// TwinCAT 3 PLC project Fraktal_Core
// Title: Fraktal_Core
// Company: fraktal-automation
// Author: fraktal-automation
// ProjectVersion: 0.1.0.3
// Description: Fraktal Core framework library: contracts, base classes (CM/EM/Unit), PermIntlk, profiler, connector base, recipe provider (Core 2.2).
// ProgramVersion: 3.1.4024.0
// libraries:
//   Tc2_Standard, * (Beckhoff Automation GmbH)
//   Tc2_System, * (Beckhoff Automation GmbH)
//   Tc2_Utilities, * (Beckhoff Automation GmbH)
//   Tc3_Module, * (Beckhoff Automation GmbH)
// project tree:
//   BaseClasses/ FB_AccessManager.TcPOU, FB_AlarmLog.TcPOU, FB_AsciiDeviceCM.TcPOU, FB_ModuleBase.TcPOU, FB_ControlModuleBase.TcPOU, FB_CycleProfiler.TcPOU, FB_CompositeModuleBase.TcPOU, FB_EquipmentModuleBase.TcPOU, FB_SequenceBase.TcPOU, FB_UnitBase.TcPOU
//   Connectivity/ FB_DeviceConnectorBase.TcPOU, FB_EcFieldbusScanner.TcPOU, FB_IoTopologyPublisher.TcPOU, FB_LocalAccessProvider.TcPOU, FB_LocalPartCarrier.TcPOU, FB_LocalRecipeProvider.TcPOU, FB_LocalStationConfig.TcPOU, FB_SimByteChannel.TcPOU, FB_TcpChannelTc3.TcPOU
//   DUTs/ E_AccessLevel.TcDUT, E_AlarmState.TcDUT, E_ByteChannelState.TcDUT, E_CarrierKind.TcDUT, E_Category.TcDUT, E_ChannelDir.TcDUT, E_ChannelKind.TcDUT, E_ExecState.TcDUT, E_FieldbusLossReaction.TcDUT, E_GatedAction.TcDUT, E_HbResult.TcDUT, E_LinkReaction.TcDUT, E_MachineState.TcDUT, E_Mode.TcDUT, E_ModeSwitchShield.TcDUT, E_PowerGroupKind.TcDUT, E_PowerState.TcDUT, E_SafetyDeviceKind.TcDUT, E_SafetyState.TcDUT, E_ModeSwitchStyle.TcDUT, E_ModuleType.TcDUT, E_NodeState.TcDUT, E_Reason.TcDUT, E_RecipeSource.TcDUT, E_ReleaseKind.TcDUT, E_ResetClass.TcDUT, E_RunStyle.TcDUT, E_Severity.TcDUT, E_StepResult.TcDUT, E_TimeClass.TcDUT, E_Verdict.TcDUT, ST_AccessPolicy.TcDUT, ST_AlarmEvent.TcDUT, ST_AlarmMeta.TcDUT, ST_BusNode.TcDUT, ST_CommandInfo.TcDUT, ST_CondRecord.TcDUT, ST_CycleProfile.TcDUT, ST_CycleSummary.TcDUT, ST_DecisionRequest.TcDUT, ST_Diagnostic.TcDUT, ST_FieldbusTopology.TcDUT, E_HmiRequestKind.TcDUT, ST_HmiRequest.TcDUT, ST_HmiResponse.TcDUT, ST_IntlkCond.TcDUT, ST_IoChannel.TcDUT, ST_IoPointIdentity.TcDUT, ST_MeasRecord.TcDUT, ST_ModePolicy.TcDUT, ST_ModelField.TcDUT, ST_ModelId.TcDUT, ST_ModuleStatus.TcDUT, ST_ControlDomainStatus.TcDUT, ST_ControlPowerStatus.TcDUT, ST_PowerGroupStatus.TcDUT, ST_SafetyDeviceStatus.TcDUT, ST_SafetyStatus.TcDUT, ST_ModuleTiming.TcDUT, ST_Nameplate.TcDUT, ST_Oee.TcDUT, ST_OeeSample.TcDUT, ST_PartContext.TcDUT, ST_PartResult.TcDUT, ST_ReleaseReason.TcDUT, ST_ReleaseReport.TcDUT, ST_StepRecord.TcDUT, ST_StepTiming.TcDUT, ST_TimingRow.TcDUT, ST_UserRecord.TcDUT, ST_TcpVisionParCfg.TcDUT, ST_TcpVisionParCmd.TcDUT, ST_TcpVisionOutCmd.TcDUT, ST_TcpVisionOutImm.TcDUT, ST_TcpCodeReaderParCfg.TcDUT, ST_TcpCodeReaderParCmd.TcDUT, ST_TcpCodeReaderOutCmd.TcDUT, ST_TcpCodeReaderOutImm.TcDUT
//   DeviceCMs/ FB_TcpCodeReaderCM.TcPOU, FB_TcpVisionCM.TcPOU
//   Interfaces/ I_AccessProvider.TcIO, I_ByteChannel.TcIO, I_ControlModule.TcIO, I_DeviceConnector.TcIO, I_EquipmentModule.TcIO, I_EventSink.TcIO, I_FieldbusScanner.TcIO, I_Module.TcIO, I_PartCarrier.TcIO, I_SequenceHost.TcIO, I_RecipeProvider.TcIO, I_StationConfig.TcIO, I_Unit.TcIO, I_VerdictProvider.TcIO
//   Params/ PL_Fraktal.TcGVL, PL_TcpDevReasons.TcGVL
//   PermIntlk/ FB_PermIntlk.TcPOU
//   Platform/ F_Now.TcPOU, F_TimingUpdate.TcPOU

// ---- DUTs/E_AccessLevel.TcDUT
// Core §7.7(a) — ordinal levels; a gated action requires CurrentLevel >= threshold
{attribute 'qualified_only'}
TYPE E_AccessLevel : (NONE := 0, OPERATOR := 1, TECHNICIAN := 2, ENGINEER := 3, ADMIN := 4) DINT;
END_TYPE

// ---- DUTs/E_AlarmState.TcDUT
// Core §8.3(b) lifecycle (ISA-18.2 mapping per §8.3(e))
{attribute 'qualified_only'}
TYPE E_AlarmState : (CLOSED := 0, ACTIVE := 1, WAIT_RESET := 2) DINT;
END_TYPE

// ---- DUTs/E_ByteChannelState.TcDUT
// Core §3.15.1a — neutral byte-transport state (non-blocking, observed over scans).
{attribute 'qualified_only'}
TYPE E_ByteChannelState : (CLOSED := 0, OPENING := 1, OPEN := 2, FAULT := 3) DINT;
END_TYPE

// ---- DUTs/E_CarrierKind.TcDUT
// Core §3.16.1
{attribute 'qualified_only'}
TYPE E_CarrierKind : (RFID := 0, DATAMATRIX := 1, BY_POSITION := 2, HOST := 3) DINT;
END_TYPE

// ---- DUTs/E_Category.TcDUT
// Core §8.8 (ST_Diagnostic.Category)
{attribute 'qualified_only'}
TYPE E_Category : (PROCESS := 0, SAFETY := 1, SYSTEM := 2) DINT;
END_TYPE

// ---- DUTs/E_ChannelDir.TcDUT
// Core §10.5.1
{attribute 'qualified_only'}
TYPE E_ChannelDir : (INPUT := 0, OUTPUT := 1) DINT;
END_TYPE

// ---- DUTs/E_ChannelKind.TcDUT
// Core §10.5.1
{attribute 'qualified_only'}
TYPE E_ChannelKind : (DIGITAL := 0, ANALOG := 1) DINT;
END_TYPE

// ---- DUTs/E_ExecState.TcDUT
// Core §6.1 — single derived command/module state
{attribute 'qualified_only'}
TYPE E_ExecState :
(
    READY   := 0,
    BUSY    := 1,
    DONE    := 2,
    ERROR   := 3,
    ABORTED := 4
) DINT;
END_TYPE

// ---- DUTs/E_FieldbusLossReaction.TcDUT
{attribute 'qualified_only'}
TYPE E_FieldbusLossReaction : (ALARM_ONLY := 0, STOP_UNIT := 1,
    POWER_GROUP_OFF := 2, CONTROL_OFF := 3) DINT;
END_TYPE

// ---- DUTs/E_GatedAction.TcDUT
// Core §7.7(a) — the enumerated protected actions (array index 0..9)
{attribute 'qualified_only'}
TYPE E_GatedAction :
(
    DATA_READ     := 0,   // view ParCfg/StationCfg values
    DATA_WRITE    := 1,   // edit ParCfg/StationCfg (§3.8a)
    MANUAL        := 2,   // manual movements default (§7.6 may raise per function)
    CHANGEOVER    := 3,   // SetModel (§3.1b)
    MODE_CHANGE   := 4,   // SetMode (§3.4)
    START_STOP    := 5,
    ALARM_HISTORY := 6,   // browse §8.3 ring
    ALARM_RESET   := 7,   // OperatorReset (§8.3(b))
    ACCESS_POLICY := 8,   // editing the policy itself
    ALARM_SHELVE  := 9,   // §8.10 shelve/unshelve an annunciated alarm
    POWER_CONTROL := 10   // §9.8 Control On/Off and power-group requests
) DINT;
END_TYPE

// ---- DUTs/E_HbResult.TcDUT
// FB_DeviceConnectorBase transport contract (Core §3.15)
{attribute 'qualified_only'}
TYPE E_HbResult : (PENDING := 0, OK := 1, FAIL := 2) DINT;
END_TYPE

// ---- DUTs/E_LinkReaction.TcDUT
// Core §3.15 — configured reaction of the fronting CM to link loss
{attribute 'qualified_only'}
TYPE E_LinkReaction : (HOLD := 0, ABORT := 1, MODE_STOP := 2) DINT;
END_TYPE

// ---- DUTs/E_MachineState.TcDUT
// Core §8.11.3 — standardized machine state for OEE, classified every scan by
// FB_UnitBase. Ordinals are a PLC↔HMI transport contract (append-only).
{attribute 'qualified_only'}
TYPE E_MachineState :
(
    PRODUCING  := 0,   // AUTO chain cycling, not blocked/starved -> uptime
    IDLE       := 1,   // ready/active outside production, no work pending
    BLOCKED    := 2,   // §8.11.1 downstream cannot accept -> external loss
    STARVED    := 3,   // §8.11.1 upstream has not delivered -> external loss
    DOWN       := 4,   // a fault holds the Unit (§8.2) -> downtime
    CHANGEOVER := 5,   // CHANGEOVER mode active (§3.4) -> planned
    STOPPED    := 6    // operator/parent Stop -> planned
) DINT;
END_TYPE

// ---- DUTs/E_Mode.TcDUT
// Core §3.4 baseline modes + §3.17 optional modes
{attribute 'qualified_only'}
TYPE E_Mode :
(
    AUTO        := 0,
    MANUAL      := 1,
    HOME        := 2,
    CHANGEOVER  := 3,
    CALIBRATION := 4,
    CAPABILITY  := 5,   // Core §3.17 (optional)
    ADJUSTMENT  := 6    // Core §3.17 (optional)
) DINT;
END_TYPE

// ---- DUTs/E_ModeSwitchShield.TcDUT
// Core §3.4.1 — may the operator leave THIS mode while its sequence runs?
{attribute 'qualified_only'}
TYPE E_ModeSwitchShield : (INTERRUPTIBLE := 0, CONFIRM := 1, BLOCKED_WHILE_RUNNING := 2) DINT;
END_TYPE

// ---- DUTs/E_PowerGroupKind.TcDUT
{attribute 'qualified_only'}
TYPE E_PowerGroupKind : (CONTROL := 0, VALVE_ZONE := 1, DRIVE_GROUP := 2,
    HEATER := 3, PROCESS_ENERGY := 4, AUXILIARY := 5) DINT;
END_TYPE

// ---- DUTs/E_PowerState.TcDUT
{attribute 'qualified_only'}
TYPE E_PowerState : (OFF := 0, ENERGIZING := 1, ON := 2,
    DEENERGIZING := 3, TRIPPED := 4, FAULT := 5) DINT;
END_TYPE

// ---- DUTs/E_SafetyDeviceKind.TcDUT
{attribute 'qualified_only'}
TYPE E_SafetyDeviceKind : (NONE := 0, ESTOP := 1, GUARD_DOOR := 2,
    LIGHT_CURTAIN := 3, SAFETY_SCANNER := 4, SAFETY_MAT := 5,
    ENABLE_SWITCH := 6, SAFETY_VALVE := 7, SAFE_DRIVE := 8,
    SAFETY_SENSOR := 9, OTHER := 10, TWO_HAND_CONTROL := 11) DINT;
END_TYPE

// ---- DUTs/E_SafetyState.TcDUT
{attribute 'qualified_only'}
TYPE E_SafetyState : (UNAVAILABLE := 0, SAFE_STATE := 1, READY := 2,
    DEMAND := 3, RESET_REQUIRED := 4, FAULT := 5) DINT;
END_TYPE

// ---- DUTs/E_ModeSwitchStyle.TcDUT
// Core §3.4.1 — how the switch completes once permitted.
{attribute 'qualified_only'}
TYPE E_ModeSwitchStyle : (GRACEFUL := 0, IMMEDIATE := 1) DINT;
END_TYPE

// ---- DUTs/E_ModuleType.TcDUT
// Core §3.2
{attribute 'qualified_only'}
TYPE E_ModuleType :
(
    NONE             := 0,
    UNIT             := 1,
    EQUIPMENT_MODULE := 2,
    CONTROL_MODULE   := 3
) DINT;
END_TYPE

// ---- DUTs/E_NodeState.TcDUT
// Core §10.5.1 — neutral fieldbus node state (EtherCAT INIT/PREOP/SAFEOP/OP map on).
// Ordinals are the HMI contract (E_NodeState in fieldbus.dart).
{attribute 'qualified_only'}
TYPE E_NodeState :
(
    OFFLINE     := 0,
    INIT        := 1,
    PREOP       := 2,
    SAFEOP      := 3,
    OPERATIONAL := 4,
    FAULT       := 5
) DINT;
END_TYPE

// ---- DUTs/E_Reason.TcDUT
// Core §8.8 — reason-code vocabulary. Framework bands only; module TYPES declare
// their band codes (10000+) as DINT constants in their own library and assign them
// to E_Reason members of ST_Diagnostic (enum is deliberately NOT 'strict' so band
// codes outside this declaration remain assignable — see IMPLEMENTATION_NOTES §3).
// Registry: Core §8.8. Codes are positive (PLCopen ErrorID is unsigned).
{attribute 'qualified_only'}
TYPE E_Reason :
(
    NONE                    := 0,

    // ── System 10–19: controller & clock health (Core §8.12, §2.7) ──
    TASK_OVERRUN            := 10,
    TASK_JITTER_HIGH        := 11,
    CPU_LOAD_HIGH           := 12,
    MEMORY_LOW              := 13,
    IPC_TEMP_HIGH           := 14,
    FIELDBUS_MASTER_FAULT   := 15,
    DC_SYNC_LOST            := 16,
    TIME_SYNC_LOST          := 17,
    UTILITY_DEVIATION       := 18,

    // ── Framework 2000–2009: common flow reasons (Core §8.8) ──
    TIMEOUT                 := 2001,
    PERMISSIVE_NOT_MET      := 2002,
    INTERLOCK_DROPPED       := 2003,
    RECIPE_INVALID          := 2004,
    STEP_STALLED            := 2005,
    RETRY_EXHAUSTED         := 2006,
    CYCLE_TIME_DEGRADED     := 2007,   // maintenance event on timing drift (Core §8.11.4(d)/§8.12)
    UNSUPPORTED_COMMAND     := 2008,   // command outside the type's supported set (§5.6)

    // ── Framework 2010–2019: external device / link supervision (Core §3.15) ──
    LINK_TIMEOUT            := 2010,
    DEVICE_NOT_READY        := 2011,
    DEVICE_PROTOCOL_ERROR   := 2012,

    // ── Framework 2020–2029: traceability / part context (Core §3.16) ──
    CARRIER_READ_FAILED     := 2020,
    CARRIER_WRITE_FAILED    := 2021,
    PART_ID_MISMATCH        := 2022,
    RESULT_RECORD_REJECTED  := 2023,
    // §3.16.3 canonical part-lifecycle events (MESSAGE ring entries, not faults)
    EVENT_PART_RECEIVED           := 2024,
    EVENT_PART_PROCESSING_STARTED := 2025,
    EVENT_PART_PROCESSED          := 2026,
    EVENT_PART_PROCESSING_ABORTED := 2027,

    // ── Framework 2900–2909: framework self-test (never raised in production) ──
    TEST_FAULT              := 2901
) DINT;
END_TYPE

// ---- DUTs/E_RecipeSource.TcDUT
// Core §3.8
{attribute 'qualified_only'}
TYPE E_RecipeSource :
(
    LOCAL       := 0,
    OPCUA       := 1,
    SOCKET_JSON := 2,
    SOCKET_XML  := 3,
    REST        := 4
) DINT;
END_TYPE

// ---- DUTs/E_ReleaseKind.TcDUT
// Core §7.8 — category of a blocking reason (for HMI grouping/icons).
{attribute 'qualified_only'}
TYPE E_ReleaseKind : (MODE := 0, ACCESS := 1, ALARM := 2, INTERLOCK := 3, OTHER := 4) DINT;
END_TYPE

// ---- DUTs/E_ResetClass.TcDUT
// Core §8.3(b) — AUTO_RESET closes when the condition re-establishes;
// MANUAL_RESET blocks (Unit will not Start) until a deliberate operator reset.
{attribute 'qualified_only'}
TYPE E_ResetClass : (AUTO_RESET := 0, MANUAL_RESET := 1) DINT;
END_TYPE

// ---- DUTs/E_RunStyle.TcDUT
// Core §3.4.2 — how a running mode advances. HOLD_TO_RUN over HMI is NON-SAFETY.
{attribute 'qualified_only'}
TYPE E_RunStyle : (CONTINUOUS := 0, SINGLE_STEP := 1, HOLD_TO_RUN := 2) DINT;
END_TYPE

// ---- DUTs/E_Severity.TcDUT
// Core §8.1
{attribute 'qualified_only'}
TYPE E_Severity : (LOW := 0, MED := 1, HIGH := 2) DINT;
END_TYPE

// ---- DUTs/E_StepResult.TcDUT
// Core §6.8/§6.10 — the shared step transition result of FB_SequenceBase.
// The ACTIVE step's action is the only writer; every chart transition reads it;
// the step's exit action clears it back to NONE (single token => no ambiguity).
// ADVANCE takes the normal successor; JUMP1..JUMP3 select declared alternative
// branches (§6.10 decisions/skips/retries) — a chart maps each to one target.
{attribute 'qualified_only'}
TYPE E_StepResult :
(
    NONE    := 0,   // stay in this step (still working/waiting)
    ADVANCE := 1,   // standard transition: the awaited work is done
    JUMP1   := 2,   // first declared alternative branch
    JUMP2   := 3,   // second declared alternative branch
    JUMP3   := 4    // third declared alternative branch
) DINT;
END_TYPE

// ---- DUTs/E_TimeClass.TcDUT
// Core §8.11.4(f) — classification of profiled time. WORK is the default; a wait
// class is declared only on genuine external waits (never to hide process slowness).
// WAIT_UPSTREAM/WAIT_DOWNSTREAM are the per-step attribution of §8.11.3 Starved/Blocked.
{attribute 'qualified_only'}
TYPE E_TimeClass :
(
    WORK            := 0,   // value-adding / process time (default)
    WAIT_UPSTREAM   := 1,   // starved: awaiting next pallet/part/material (§8.11.3)
    WAIT_DOWNSTREAM := 2,   // blocked: awaiting outfeed / downstream take-over (§8.11.3)
    WAIT_OPERATOR   := 3,   // §6.11 decision / manual intervention
    WAIT_EXTERNAL   := 4    // host/MES/tool response (§3.15, §11.6)
) DINT;
END_TYPE

// ---- DUTs/E_Verdict.TcDUT
// Core §3.16.1
{attribute 'qualified_only'}
TYPE E_Verdict : (NONE := 0, OK := 1, NOK := 2, REWORK := 3) DINT;
END_TYPE

// ---- DUTs/ST_AccessPolicy.TcDUT
// Core §7.7(b) — per-station required level per action. SHIPPED DEFAULT: fully open
// (NONE everywhere) — locking down is a deliberate deployment decision, reviewed at
// commissioning (§14). Held as persistent station configuration (§3.8a).
TYPE ST_AccessPolicy :
STRUCT
    Required       : ARRAY[0..10] OF E_AccessLevel;  // index = TO_INT(E_GatedAction)
    SessionTimeout : TIME := T#0S;                   // idle auto-logout; T#0S = never
END_STRUCT
END_TYPE

// ---- DUTs/ST_AlarmEvent.TcDUT
// Core §8.3(a) — one alarm/event with full lifecycle. Same reason vocabulary as
// every diagnostic (§8.8): the event IS the diagnostic plus lifecycle.
TYPE ST_AlarmEvent :
STRUCT
    ReasonCode  : E_Reason;
    Description : STRING(255);
    SourcePath  : STRING(255);   // module browse path (§4.8) = historian tag path
    IoTag       : STRING(80);    // exact implicated electrical tag; untranslated
    IoAddress   : STRING(80);    // terminal/channel locator
    Severity    : E_Severity;
    Category    : E_Category;
    ResetClass  : E_ResetClass;
    State       : E_AlarmState;
    ComeAt      : DT;            // synchronized stamps (§2.7)
    GoneAt      : DT;
    ResetAt     : DT;            // MANUAL_RESET only
    Duration    : TIME;          // monotonic come->gone (§8.11.4(e) two-clock rule)
    Shelved     : BOOL;          // §8.10 annunciation suppressed (control unaffected)
    ShelvedUntil: DT;            // display only; enforcement is the log's countdown
END_STRUCT
END_TYPE

// ---- DUTs/ST_AlarmMeta.TcDUT
// Core §8.9 — runtime rationalization record for one ReasonCode: what the operator
// should DO, what happens if they don't, and whether shelving is permitted.
TYPE ST_AlarmMeta :
STRUCT
    ReasonCode     : E_Reason;
    OperatorAction : STRING(255);  // "what do I do about this?"
    Consequence    : STRING(255);
    Shelvable      : BOOL;         // §8.10: no record or FALSE -> not shelvable
END_STRUCT
END_TYPE

// ---- DUTs/ST_BusNode.TcDUT
// Core §10.5.1 — one fieldbus node. The node/channel arrays are populated at
// runtime from the master's diagnostics (TC3 §10.6: EtherCAT/ADS); this is the
// published shape the generic HMI renders. Children are referenced by index into
// the master's flat node table to keep the DUT bounded (no recursion in IEC types).
TYPE ST_BusNode :
STRUCT
    Name        : STRING(80);
    DescriptionKey : STRING(160); // hardware-description localization key
    TypeId      : STRING(80);   // vendor/product
    Address     : STRING(40);   // topological + logical
    State       : E_NodeState;
    LinkOk      : BOOL;
    ParentIdx   : INT;          // index of parent node in the flat table (0 = root)
    ChannelCount: INT;
    Channels    : ARRAY[1..PL_Fraktal.MAX_NODE_CHANNELS] OF ST_IoChannel;
END_STRUCT
END_TYPE

// ---- DUTs/ST_CommandInfo.TcDUT
// Core §7.6.1 — one entry in a module's self-describing command catalog.
// Value is what ExecuteCommand accepts (§3.2); Label is the button text.
TYPE ST_CommandInfo :
STRUCT
    Value : DINT;
    Label : STRING(120);   // localization key; resolved by the HMI catalog
END_STRUCT
END_TYPE

// ---- DUTs/ST_CondRecord.TcDUT
// Core §6.9(b) — named plain-condition wait
TYPE ST_CondRecord :
STRUCT
    Label : STRING(120);   // localization key
    Ok    : BOOL;
END_STRUCT
END_TYPE

// ---- DUTs/ST_CycleProfile.TcDUT
// Core §8.11.4(b)/(f) — one completed cycle: ordered waterfall + time-class split.
// ByClass is indexed by TO_INT(E_TimeClass): 0=WORK 1=WAIT_UPSTREAM 2=WAIT_DOWNSTREAM
// 3=WAIT_OPERATOR 4=WAIT_EXTERNAL.
TYPE ST_CycleProfile :
STRUCT
    CycleNo   : UDINT;
    Started   : DT;
    Total     : TIME;     // reconciles with the §8.11.1 CycleTime
    WorkTime  : TIME;     // §8.11.4(f): THE REAL CYCLE TIME (= ByClass[WORK])
    WaitTime  : TIME;     // Total - WorkTime (all wait classes)
    ByClass   : ARRAY[0..4] OF TIME;
    NSteps    : INT;
    Truncated : BOOL;     // more step changes than MAX_PROFILE_STEPS
    Steps     : ARRAY[1..PL_Fraktal.MAX_PROFILE_STEPS] OF ST_StepTiming;
END_STRUCT
END_TYPE

// ---- DUTs/ST_CycleSummary.TcDUT
// Core §8.11.4 — one completed cycle's totals for the trend ring: enough to chart
// WHY cycle time moved (work vs each wait class) without the full step waterfall.
TYPE ST_CycleSummary :
STRUCT
    CycleNo  : UDINT;
    Started  : DT;                    // synchronized wall clock (Core §2.7)
    Total    : TIME;
    WorkTime : TIME;                  // §8.11.4(f) — the real cycle time
    WaitTime : TIME;
    ByClass  : ARRAY[0..4] OF TIME;   // indexed by TO_INT(E_TimeClass)
END_STRUCT
END_TYPE

// ---- DUTs/ST_DecisionRequest.TcDUT
// Core §6.11 — typed operator decision request
TYPE ST_DecisionRequest :
STRUCT
    Prompt     : STRING(255);   // localization key; Options[] are keys too
    Options    : ARRAY[1..PL_Fraktal.MAX_OPTIONS] OF STRING(64);
    Default    : INT;            // option index applied on timeout
    Timeout    : TIME;           // T#0S = wait indefinitely
    SourcePath : STRING(255);    // raising module (Core §4.8)
END_STRUCT
END_TYPE

// ---- DUTs/ST_Diagnostic.TcDUT
// Core §8.8 — the full first-out reason record
TYPE ST_Diagnostic :
STRUCT
    ReasonCode  : E_Reason;      // named reason; ErrorID = TO_DWORD(ReasonCode)
    SourcePath  : STRING(255);   // OPC UA browse path of the module/condition (Core §4.8)
    Description : STRING(255);   // localization key (from PermIntlk or module); never operator prose
    IoTag       : STRING(80);    // untranslated schematic/electrical tag of implicated channel
    IoAddress   : STRING(80);    // terminal/channel locator, e.g. EL1809 Ch5
    Severity    : E_Severity;    // LOW | MED | HIGH (Core §8.1)
    Category    : E_Category;    // PROCESS | SAFETY | SYSTEM
    Since       : DT;            // first-out timestamp (synchronized clock, Core §2.7)
END_STRUCT
END_TYPE

// ---- DUTs/ST_FieldbusTopology.TcDUT
// Core §10.5.1 — bounded published fieldbus table plus mapping validation.
// Physical discovery fills nodes; the project catalog joins approved I/O metadata.
TYPE ST_FieldbusTopology :
STRUCT
    NodeCount : INT;
    Nodes : ARRAY[1..PL_Fraktal.MAX_BUS_NODES] OF ST_BusNode;
    MappingValid : BOOL;
    MappingDiagnostic : STRING(255); // localization key; empty when valid
END_STRUCT
END_TYPE

// ---- DUTs/E_HmiRequestKind.TcDUT
// Core §3.10/§14 — generic OPC UA request mailbox operation.
// Append-only: ordinal values are a transport contract with every HMI adapter.
{attribute 'qualified_only'}
TYPE E_HmiRequestKind :
(
    NONE             := 0,
    LOGIN            := 1,
    LOGOUT           := 2,
    SET_MODE         := 3,
    SET_MODEL        := 4,
    START            := 5,
    STOP             := 6,
    CONTROL_ON       := 7,
    CONTROL_OFF      := 8,
    OPERATOR_RESET   := 9,
    DECISION_ANSWER  := 10,
    MANUAL_COMMAND   := 11,
    SET_RUN_STYLE    := 12,
    STEP_REQUEST     := 13,
    SET_HOLD_RUN     := 14,
    RELEASE_START    := 15,
    RELEASE_MANUAL   := 16,
    RELEASE_ACTION   := 17,
    RESET_OEE        := 18,
    WRITE_CONFIG     := 19,
    SHELVE_ALARM     := 20,
    UNSHELVE_ALARM   := 21,
    FORCE_CHANNEL    := 22
) DINT;
END_TYPE

// ---- DUTs/ST_HmiRequest.TcDUT
// Core §3.10/§14 — write-only-by-convention generic Unit request mailbox.
// The client writes all arguments first and Sequence LAST as the atomic commit marker.
TYPE ST_HmiRequest :
STRUCT
    Kind       : E_HmiRequestKind;
    TargetPath : STRING(255);
    NameValue  : STRING(160);
    TextValue  : STRING(255);
    User       : STRING(32);
    Secret     : STRING(32);   // base clears immediately after sampling
    IntValue   : DINT;
    BoolValue  : BOOL;
    DurationMs : UDINT;
    Sequence   : UDINT;        // monotonically changing commit marker
END_STRUCT
END_TYPE

// ---- DUTs/ST_HmiResponse.TcDUT
// Core §3.10/§14 — acknowledgement for ST_HmiRequest.
TYPE ST_HmiResponse :
STRUCT
    AckSequence : UDINT;
    Accepted    : BOOL;           // request acted or query completed
    Diagnostic  : STRING(255);    // localization key when refused/unsupported
    Report      : ST_ReleaseReport;
END_STRUCT
END_TYPE

// ---- DUTs/ST_IntlkCond.TcDUT
// Core §7.2 — per-condition record of FB_PermIntlk
TYPE ST_IntlkCond :
STRUCT
    Defined     : BOOL;
    Description : STRING(255);   // localization key
    Reason      : E_Reason;
    Bypassable  : BOOL;
END_STRUCT
END_TYPE

// ---- DUTs/ST_IoChannel.TcDUT
// Core §10.5.1 — one fieldbus I/O channel (published for the topology view §3.13)
TYPE ST_IoChannel :
STRUCT
    Name       : STRING(80);
    DescriptionKey : STRING(160); // project/standard localization key
    Address    : STRING(80);    // physical locator, e.g. EL1809 Ch5
    Path       : STRING(255);   // unique channel path (force/audit identity)
    ModulePath : STRING(255);   // owning module browse path for cross-navigation
    Dir        : E_ChannelDir;
    Kind       : E_ChannelKind;
    BoolValue  : BOOL;          // digital
    AnalogValue: REAL;          // analog (scaled)
    Unit       : STRING(16);
    Forced     : BOOL;
    Quality    : BOOL;          // TRUE = good
    FaultActive: BOOL;          // a module diagnostic implicates this exact channel
    Diagnostic : STRING(255);   // localization key; Name remains the exact I/O tag
END_STRUCT
END_TYPE

// ---- DUTs/ST_IoPointIdentity.TcDUT
// Core §10.2/§10.5.1 — immutable engineering identity of one mapped I/O point.
// Device types consume roles; the project catalog supplies this physical identity.
TYPE ST_IoPointIdentity :
STRUCT
    Tag : STRING(80);
    Address : STRING(80);
    DescriptionKey : STRING(160);
    Path : STRING(255);
    ModulePath : STRING(255);
END_STRUCT
END_TYPE

// ---- DUTs/ST_MeasRecord.TcDUT
// Core §3.16.1 — one measured value with limits and a FIXED engineering unit (Core §3.8)
TYPE ST_MeasRecord :
STRUCT
    Name   : STRING(64);
    Value  : LREAL;
    Minimum : LREAL;
    Maximum : LREAL;
    Target : LREAL;
    Unit   : STRING(16);   // fixed engineering unit — not runtime-variable (Core §3.8)
    InTol  : BOOL;
END_STRUCT
END_TYPE

// ---- DUTs/ST_ModePolicy.TcDUT
// Core §3.4.1 — per-mode switch policy, indexed by TO_INT(E_Mode). Station config
// (§3.8a): editable per deployment, sensible defaults set in FB_UnitBase init.
TYPE ST_ModePolicy :
STRUCT
    Shield : E_ModeSwitchShield;
    Style  : E_ModeSwitchStyle;
END_STRUCT
END_TYPE

// ---- DUTs/ST_ModelField.TcDUT
// Core §3.8a — one client-defined named model field
TYPE ST_ModelField : STRUCT  Name : STRING(32);  Value : STRING(64);  END_STRUCT END_TYPE

// ---- DUTs/ST_ModelId.TcDUT
// Core §3.1b/§3.8a — a root Unit's active model identity (the changeover KEY).
// Two roots may hold different ST_ModelId simultaneously (§3.1b).
TYPE ST_ModelId :
STRUCT
    ModelCode : STRING(64);   // minimum required identity
    Family    : STRING(64);   // optional
    Variant   : STRING(64);   // optional
    Fields    : ARRAY[1..PL_Fraktal.MAX_MODEL_FIELDS] OF ST_ModelField;  // optional client fields
    NField    : INT;
END_STRUCT
END_TYPE

// ---- DUTs/ST_ModuleStatus.TcDUT
// Core §3.10(a')/§3.12/§6.9(a) — the DATA MIRROR every module publishes each scan.
// Properties/methods serve PLC code; this struct serves OPC UA/HMI. It is the
// framework baseline of the OutImm role: name, tier, state summary, and the live
// first-out diagnostic — everything a generic tile needs, browsable by type.
TYPE ST_ModuleStatus :
STRUCT
    Name        : STRING(80);     // = browse name (§4.8) — the tile caption
    DisplayNameKey : STRING(160); // optional localization key; Name remains identity
    DescriptionKey : STRING(160); // optional module information localization key
    ModuleType  : E_ModuleType;   // UNIT | EQUIPMENT_MODULE | CONTROL_MODULE (tile kind)
    State       : E_ExecState;    // the tile state LED
    FaultActive : BOOL;
    Diagnostic  : ST_Diagnostic;  // live first-out (§6.9(a)) — the tile message line
    TileEnable  : BOOL := TRUE;   // §3.13: render as a tile on the parent's child view
    ControlDomainId : STRING(80); // §9.8: '' = no safety/control-power arrangement
END_STRUCT
END_TYPE

// ---- DUTs/ST_ControlDomainStatus.TcDUT
// Core §9.8 — one independently owned safety/control-power arrangement.
// A Unit consumes this record; zero or many Units may reference the same domain.
TYPE ST_ControlDomainStatus :
STRUCT
    Present         : BOOL;        // FALSE = this Unit has no assigned control domain
    Id              : STRING(80);  // stable deployment identity, not a Unit browse path
    Name            : STRING(80);  // operator-facing cage/cell/energy-area name
    ReadyForStart   : BOOL;        // coordinator aggregate; fail-closed when Present
    Safety          : ST_SafetyStatus;
    ControlPower    : ST_ControlPowerStatus;
    MemberCount     : INT;
    MemberUnitPaths : ARRAY[1..PL_Fraktal.MAX_CONTROL_DOMAIN_UNITS] OF STRING(255);
END_STRUCT
END_TYPE

// ---- DUTs/ST_ControlPowerStatus.TcDUT
TYPE ST_ControlPowerStatus :
STRUCT
    Present        : BOOL;
    RequestedOn    : BOOL;
    ControlOn      : BOOL;
    Transitioning  : BOOL;
    RearmRequired  : BOOL;
    GroupCount     : INT;
    Groups         : ARRAY[1..PL_Fraktal.MAX_POWER_GROUPS] OF ST_PowerGroupStatus;
    Diagnostic     : ST_Diagnostic;
END_STRUCT
END_TYPE

// ---- DUTs/ST_PowerGroupStatus.TcDUT
TYPE ST_PowerGroupStatus :
STRUCT
    Present              : BOOL;
    Name                 : STRING(80);
    Kind                 : E_PowerGroupKind;
    State                : E_PowerState;
    RequiredForControl   : BOOL;
    RequestedOn          : BOOL;
    PowerOn              : BOOL;
    SafetyPermit         : BOOL;
    FieldbusHealthy      : BOOL;
    FieldbusLossReaction : E_FieldbusLossReaction;
    RearmRequired        : BOOL;
    Diagnostic           : ST_Diagnostic;
END_STRUCT
END_TYPE

// ---- DUTs/ST_SafetyDeviceStatus.TcDUT
TYPE ST_SafetyDeviceStatus :
STRUCT
    Present           : BOOL;
    Name              : STRING(80);
    Kind              : E_SafetyDeviceKind;
    State             : E_SafetyState;
    Ready             : BOOL;
    DemandActive      : BOOL;
    SafeStateActive   : BOOL;
    ResetRequired     : BOOL;
    FaultActive       : BOOL;
    MutingActive      : BOOL;   // safety-evaluated; standard PLC cannot set
    BridgeActive      : BOOL;   // keyed safety bridge; read-only here
    FieldbusHealthy   : BOOL;
    AffectedPowerMask : DWORD;  // documentation/status mapping, never safety logic
    Description       : STRING(255);   // localization key
END_STRUCT
END_TYPE

// ---- DUTs/ST_SafetyStatus.TcDUT
TYPE ST_SafetyStatus :
STRUCT
    Present         : BOOL;
    AllSafe         : BOOL;
    DemandActive    : BOOL;
    ResetRequired   : BOOL;
    FaultActive     : BOOL;
    MutingActive    : BOOL;
    BridgeActive    : BOOL;
    StopRequested   : BOOL;
    DeviceCount     : INT;
    Devices         : ARRAY[1..PL_Fraktal.MAX_SAFETY_DEVICES] OF ST_SafetyDeviceStatus;
END_STRUCT
END_TYPE

// ---- DUTs/ST_ModuleTiming.TcDUT
// Core §8.11.4(a) — per-module command timing, maintained by FB_ControlModuleBase.
// Fixed-size; capture never allocates at runtime (Core §8.11.4(e)).
TYPE ST_ModuleTiming :
STRUCT
    LastCmdTime : TIME;   // duration of the most recently completed command
    Rows        : ARRAY[1..PL_Fraktal.MAX_CMD_STATS] OF ST_TimingRow;
    Truncated   : BOOL;   // more distinct command ids than MAX_CMD_STATS
END_STRUCT
END_TYPE

// ---- DUTs/ST_Nameplate.TcDUT
// Core §3.10.1 — digital nameplate (asset identity). Field set aligned with the
// IDTA 02006 Digital Nameplate submodel so the AAS projection (Annex K) is direct.
// Static identity: set once at Setup, never runtime-mutated, never HMI-writable.
TYPE ST_Nameplate :
STRUCT
    ProductUri        : STRING(255);  // globally unique asset URI (IDTA: URIOfTheProduct)
    ManufacturerName  : STRING(80);
    ProductDesignation: STRING(80);
    SerialNumber      : STRING(40);
    YearOfConstruction: STRING(8);
    HardwareVersion   : STRING(24);
    FirmwareVersion   : STRING(24);
    SoftwareVersion   : STRING(24);
    OrderCode         : STRING(40);
    DocumentationUrl  : STRING(255);  // manual / handover docs (cf. IDTA 02004)
END_STRUCT
END_TYPE

// ---- DUTs/ST_Oee.TcDUT
// Core §8.5.1 — OEE snapshot + accumulators (published; derived, never lies).
// Factors are 0..1 REAL; a factor with Valid=FALSE is omitted from Oee, not 100%.
TYPE ST_Oee :
STRUCT
    RunMs        : UDINT;   // time buckets since reset (ms; wraps ~49 days)
    DownMs       : UDINT;
    IdleMs       : UDINT;
    Availability : REAL;    AvailValid : BOOL;
    Performance  : REAL;    PerfValid  : BOOL;   // needs IdealCycleMs > 0
    Quality      : REAL;    QualValid  : BOOL;
    Oee          : REAL;    OeeValid   : BOOL;   // product of the VALID factors only
    IdealCycleMs : UDINT;   // §3.8 per-model config; 0 = performance not computed
END_STRUCT
END_TYPE

// ---- DUTs/ST_OeeSample.TcDUT
// Core §8.5.1 — one trend sample for the HMI sparkline ring.
TYPE ST_OeeSample :
STRUCT
    Availability : REAL;
    Performance  : REAL;
    Quality      : REAL;
    Oee          : REAL;
    OeeValid     : BOOL;
END_STRUCT
END_TYPE

// ---- DUTs/ST_PartContext.TcDUT
// Core §3.16.1
TYPE ST_PartContext :
STRUCT
    Uid         : STRING(64);    // serial / unique id ('' if no part)
    Present     : BOOL;
    CarrierKind : E_CarrierKind;
    Result      : ST_PartResult;
    Parents     : ARRAY[1..PL_Fraktal.MAX_GENEALOGY] OF STRING(64);
END_STRUCT
END_TYPE

// ---- DUTs/ST_PartResult.TcDUT
// Core §3.16.1
TYPE ST_PartResult :
STRUCT
    Verdict     : E_Verdict;     // NONE | OK | NOK | REWORK
    ReasonCode  : E_Reason;      // first NOK reason — SAME vocabulary as a fault (Core §8.8)
    Records     : ARRAY[1..PL_Fraktal.MAX_RESULTS] OF ST_MeasRecord;
    StationPath : STRING(255);   // browse path of the producing station (Core §4.8)
    Stamp       : DT;            // synchronized timestamp (Core §2.7)
END_STRUCT
END_TYPE

// ---- DUTs/ST_ReleaseReason.TcDUT
// Core §7.8 — one unmet precondition in a release report.
TYPE ST_ReleaseReason :
STRUCT
    Description : STRING(255);   // localization key
    ReasonCode  : E_Reason;
    SourcePath  : STRING(255);   // qualified module identity that owns the condition
    Kind        : E_ReleaseKind;
    Bypassable  : BOOL;      // §7.4 — this interlock may be bypassed
END_STRUCT
END_TYPE

// ---- DUTs/ST_ReleaseReport.TcDUT
// Core §7.8 — the full 'why is this blocked?' rollup, published for the HMI.
// Complete by contract: lists EVERY failing precondition, not just first-out.
TYPE ST_ReleaseReport :
STRUCT
    Released : BOOL;         // TRUE = nothing blocks (Count = 0)
    Count    : INT;
    Reasons  : ARRAY[1..PL_Fraktal.MAX_RELEASE_REASONS] OF ST_ReleaseReason;
END_STRUCT
END_TYPE

// ---- DUTs/ST_StepRecord.TcDUT
// Core §6.5 — what the stall walk reads
TYPE ST_StepRecord :
STRUCT
    StepNo        : INT;
    StepName      : STRING(120);   // localization key
    AwaitingLabel : STRING(120);   // e.g. 'ClampStation.CLAMP' ('' if none)
    Class         : E_TimeClass;   // Core §8.11.4(f) — WORK unless a genuine wait
    ExpectedTime  : TIME;          // defaults from the awaited command's timeout
    Conds         : ARRAY[1..PL_Fraktal.MAX_STEP_CONDS] OF ST_CondRecord;
END_STRUCT
END_TYPE

// ---- DUTs/ST_StepTiming.TcDUT
// Core §8.11.4(b)/(f) — one step of a cycle profile (Gantt/waterfall row)
TYPE ST_StepTiming :
STRUCT
    StepNo   : INT;
    StepName : STRING(120);   // localization key
    Class    : E_TimeClass;  // WORK unless the step declared a wait class (§8.11.4(f))
    Started  : DT;           // synchronized wall clock (Core §2.7) — aligns across stations
    Duration : TIME;         // monotonic-clock duration (TC3 §8.11)
    Expected : TIME;         // §8.11.4(c) — the step's declared guard, drawn vs actual (0 = none)
END_STRUCT
END_TYPE

// ---- DUTs/ST_TimingRow.TcDUT
// Core §8.11.4 — one timing aggregate, keyed by command id (a) or StepNo (b)
TYPE ST_TimingRow :
STRUCT
    Id    : DINT;         // TO_DINT(E_<Type>Command) or StepNo; 0 = untagged
    Label : STRING(120);   // command/step localization key for the HMI table
    Class : E_TimeClass;  // §8.11.4(f); commands are WORK by definition
    Count : UDINT;        // completed executions (0 = row unused)
    Last  : TIME;
    Minimum : TIME;
    Maximum : TIME;
    Avg   : TIME;         // running mean (F_TimingUpdate)
END_STRUCT
END_TYPE

// ---- DUTs/ST_UserRecord.TcDUT
// Core §7.7(c) — FB_LocalAccessProvider table entry (local default; server-side
// auth substitutes via I_AccessProvider without touching module code)
TYPE ST_UserRecord :
STRUCT
    User  : STRING(32);
    Pin   : STRING(32);
    Level : E_AccessLevel;
END_STRUCT
END_TYPE

// ---- DUTs/ST_TcpVisionParCfg.TcDUT
TYPE ST_TcpVisionParCfg :
STRUCT
    SchemaVersion : UINT := 1;
    Host          : STRING(80);
    Port          : UINT;
    Terminator    : STRING(2) := '$R';
    RespTimeout   : TIME := T#2S;
    TriggerCmd    : STRING(40) := 'T';
    OkPrefix      : STRING(20) := 'OK';
    NgPrefix      : STRING(20) := 'NG';
    ResultSep     : STRING(2) := ',';
END_STRUCT
END_TYPE

// ---- DUTs/ST_TcpVisionParCmd.TcDUT
TYPE ST_TcpVisionParCmd :
STRUCT
    Reserved : BOOL;
END_STRUCT
END_TYPE

// ---- DUTs/ST_TcpVisionOutCmd.TcDUT
TYPE ST_TcpVisionOutCmd :
STRUCT
    JudgeOk   : BOOL;
    ResultData: STRING(255);
END_STRUCT
END_TYPE

// ---- DUTs/ST_TcpVisionOutImm.TcDUT
TYPE ST_TcpVisionOutImm :
STRUCT
    LinkState    : E_ByteChannelState;
    LastResponse : STRING(255);
    Diagnostic   : ST_Diagnostic;
END_STRUCT
END_TYPE

// ---- DUTs/ST_TcpCodeReaderParCfg.TcDUT
TYPE ST_TcpCodeReaderParCfg :
STRUCT
    SchemaVersion : UINT := 1;
    Host          : STRING(80);
    Port          : UINT;
    Terminator    : STRING(2) := '$R';
    RespTimeout   : TIME := T#2S;
    TriggerCmd    : STRING(40) := 'T';
    NoReadText    : STRING(40) := 'NOREAD';
END_STRUCT
END_TYPE

// ---- DUTs/ST_TcpCodeReaderParCmd.TcDUT
TYPE ST_TcpCodeReaderParCmd :
STRUCT
    MatchCode : STRING(255);
END_STRUCT
END_TYPE

// ---- DUTs/ST_TcpCodeReaderOutCmd.TcDUT
TYPE ST_TcpCodeReaderOutCmd :
STRUCT
    Code    : STRING(255);
    NoRead  : BOOL;
    MatchOk : BOOL;
END_STRUCT
END_TYPE

// ---- DUTs/ST_TcpCodeReaderOutImm.TcDUT
TYPE ST_TcpCodeReaderOutImm :
STRUCT
    LinkState    : E_ByteChannelState;
    LastResponse : STRING(255);
    Diagnostic   : ST_Diagnostic;
END_STRUCT
END_TYPE

// ---- Params/PL_Fraktal.TcGVL
{attribute 'qualified_only'}
// Fraktal Core — framework constants (Core §7.2, §3.2, §6.5, §3.16, §6.11)
VAR_GLOBAL CONSTANT
    MAX_PERMINTLK_COND   : INT := 16;   // Core §7.2 (default 16)
    MAX_EM_CHILDREN      : INT := 16;   // Core §3.2 / §8.2
    MAX_STEP_CONDS       : INT := 8;    // Core §6.9(b) condition records per step
    MAX_GENEALOGY        : INT := 8;    // Core §3.16.1
    MAX_RESULTS          : INT := 32;   // Core §3.16.1
    MAX_OPTIONS          : INT := 6;    // Core §6.11
    MAX_CMD_STATS        : INT := 8;    // Core §8.11.4(a) — distinct command ids per module
    MAX_PROFILE_STEPS    : INT := 32;   // Core §8.11.4(b) — steps per cycle profile
    MAX_RECIPES          : INT := 16;   // Core §3.8 — records per FB_LocalRecipeProvider
    MAX_MODEL_FIELDS     : INT := 8;    // Core §3.8a — client-defined named model fields
    MAX_STATIONCFG       : INT := 16;   // Core §3.8a — records per FB_LocalStationConfig
    MAX_ALARM_ACTIVE     : INT := 16;   // Core §8.3 — concurrently open events per Unit
    MAX_ALARM_RING       : INT := 64;   // Core §8.3 — closed-event history ring per Unit
    MAX_USERS            : INT := 16;   // Core §7.7 — FB_LocalAccessProvider user table
    MAX_POS_SENSORS      : INT := 2;    // redundant sensors per cylinder position (duplex; raise for 2oo3)
    MAX_NODE_CHANNELS    : INT := 16;   // Core §10.5.1 — I/O channels per fieldbus node
    MAX_BUS_NODES        : INT := 64;   // Core §10.5.1 — nodes in the flat topology table
    MAX_CMD_CATALOG      : INT := 12;   // Core §7.6.1 — manual commands a module may publish
    MODE_COUNT           : INT := 7;    // Core §3.4 — E_Mode entries (AUTO..ADJUSTMENT), for policy array
    MAX_RELEASE_REASONS  : INT := 24;   // Core §7.8 — entries in a release report
    MAX_OEE_SAMPLES      : INT := 60;      // Core §8.5.1 — trend ring length
    MAX_CYCLE_HISTORY    : INT := 60;      // Core §8.11.4 — per-cycle summary ring (trend charts)
    OEE_SAMPLE_MS        : UDINT := 60000; // Core §8.5.1 — sample period (1 min)
    MAX_ALARM_META       : INT := 32;      // Core §8.9 — rationalization records per log
    MAX_SHELF_S          : UDINT := 28800; // Core §8.10 — shelf cap (8h)
    MAX_DIAG_RING        : INT := 16;   // Core §6.9(a) — Unit diagnostic history depth
    MAX_SAFETY_DEVICES   : INT := 16;   // Core §9 — published safety aliases per module/zone
    MAX_POWER_GROUPS     : INT := 8;    // Core §9 — independently controlled energy groups
    MAX_CONTROL_DOMAIN_UNITS : INT := 16; // Core §9.8 — root Units sharing one arrangement
END_VAR

// ---- Params/PL_TcpDevReasons.TcGVL
// Core §3.15.1a / §8.8 — TCP/ASCII device CM base band 10401-10406 (registered).
// Device profiles extend within 10401-10499.
{attribute 'qualified_only'}
VAR_GLOBAL CONSTANT
    DEV_CHANNEL_FAULT : DINT := 10401;   // transport reported FAULT
    DEV_RESP_TIMEOUT  : DINT := 10402;   // no terminated response within RespTimeout
    DEV_PROTOCOL      : DINT := 10403;   // profile parse rejected the response
    DEV_NOT_CONNECTED : DINT := 10404;   // request issued while channel not OPEN
    DEV_CFG_INVALID   : DINT := 10405;   // missing host/port/channel at Setup
    DEV_RX_OVERFLOW   : DINT := 10406;   // response exceeded the RX buffer
END_VAR

// ---- Interfaces/I_AccessProvider.TcIO
// Core §7.7(c) — credential validation, injectable like every provider (§3.8).
// Returns the granted level; NONE = authentication failed.
INTERFACE I_AccessProvider

METHOD Authenticate : E_AccessLevel
VAR_INPUT
    User   : STRING(32);
    Secret : STRING(32);
END_VAR
END_METHOD

END_INTERFACE

// ---- Interfaces/I_ByteChannel.TcIO
// Core §3.15.1a — THE porting seam for TCP/serial devices. Non-blocking,
// cyclic-poll semantics: every method returns immediately; progress is observed
// via State() over scans. [TC3]: Tc2_TcpIp (TC3 §3.15); CODESYS: SysSocket/NBS;
// Siemens: TSEND_C/TRCV_C wrappers. Device CMs written against this interface
// port between PLC brands unmodified (O4/O8).
INTERFACE I_ByteChannel

// begin opening (non-blocking); observe State() -> OPENING -> OPEN/FAULT
METHOD Open : BOOL
VAR_INPUT
    Host : STRING(80);
    Port : UINT;
END_VAR
END_METHOD

METHOD Close : BOOL
END_METHOD

// queue Text for transmission (no terminator added here). FALSE if not OPEN.
METHOD Send : BOOL
VAR_INPUT
    Text : STRING(255);
END_VAR
END_METHOD

// drain received bytes: appends to Buffer, returns chars appended this call.
METHOD Poll : INT
VAR_IN_OUT
    Buffer : STRING(255);
END_VAR
END_METHOD

METHOD State : E_ByteChannelState
END_METHOD

// drive the channel's internal state machine once per scan
METHOD Tick : BOOL
END_METHOD

END_INTERFACE

// ---- Interfaces/I_ControlModule.TcIO
// Core §3.2 — HAL-bound leaf tier. Same generic command vocabulary as I_EquipmentModule.
INTERFACE I_ControlModule EXTENDS I_Module

METHOD ExecuteCommand : BOOL
VAR_INPUT
    Command : DINT;   // value of the type's E_<Type>Command
END_VAR
END_METHOD

METHOD AbortCommand : BOOL
END_METHOD

END_INTERFACE

// ---- Interfaces/I_DeviceConnector.TcIO
// Core §3.15 — networked smart device: session + mandatory link supervision.
INTERFACE I_DeviceConnector EXTENDS I_Module

METHOD Connect : BOOL
END_METHOD

METHOD Disconnect : BOOL
END_METHOD

// timestamp of last healthy heartbeat (Core §2.7)
PROPERTY LastSeen : DT
GET
END_GET
END_PROPERTY

// session up AND heartbeat healthy (Core §3.15.2)
PROPERTY Linked : BOOL
GET
END_GET
END_PROPERTY

// first-out link/protocol reason when not Linked
PROPERTY LinkReason : ST_Diagnostic
GET
END_GET
END_PROPERTY

END_INTERFACE

// ---- Interfaces/I_EquipmentModule.TcIO
// Core §3.2 — discrete-command tier. Generic command id is DINT (a per-type
// E_<Type>Command enum cannot appear in a shared interface); the type's typed
// PLCopen surface (Command input) remains primary. IMPLEMENTATION_NOTES §2.
INTERFACE I_EquipmentModule EXTENDS I_Module

METHOD ExecuteCommand : BOOL
VAR_INPUT
    Command : DINT;   // value of the type's E_<Type>Command
END_VAR
END_METHOD

METHOD AbortCommand : BOOL
END_METHOD

END_INTERFACE

// ---- Interfaces/I_EventSink.TcIO
// Core §8.3(d) — historian/database adapter hook. Invoked at come and at close;
// implementations (OPC UA A&C, SQL, MES) are deployment choices — deferred by design.
INTERFACE I_EventSink

METHOD OnEvent : BOOL
VAR_INPUT
    Ev : ST_AlarmEvent;
END_VAR
END_METHOD

END_INTERFACE

// ---- Interfaces/I_FieldbusScanner.TcIO
// Core §10.5.1 / TC3 §10.6 — the seam an integrator implements to populate the
// fieldbus topology model from a real master's diagnostics. The application owns
// the flat node table; the scanner fills it each refresh and answers force writes.
// A default EtherCAT implementation is FB_EcFieldbusScanner (skeleton). Other buses
// (PROFINET, EtherNet/IP gateways) implement this same interface (O4/O8).
INTERFACE I_FieldbusScanner

// Rebuild the node table from the master; returns node count (0 = master down).
// Fills Nodes[1..count] (ParentIdx/State/Channels). Called at a slow cadence
// (e.g. 200 ms) — topology changes rarely; live values refresh separately.
METHOD Scan : INT
VAR_IN_OUT
    Data : ST_FieldbusTopology;
END_VAR
END_METHOD

// Update only the live channel values/quality of an already-scanned table (fast
// cadence, every scan). Keeps topology stable while values move.
METHOD RefreshValues : BOOL
VAR_IN_OUT
    Data : ST_FieldbusTopology;
END_VAR
END_METHOD

// Apply/clear an OUTPUT force on one channel (Core §10.5.1, output-only rule).
// MUST already be authorized by the caller (§7.6/§7.7); the scanner only performs
// the write and returns success (FALSE if the channel is an INPUT or unknown).
// Writes the mapped OUTPUT variable through the application — never a raw
// process-image force, never an input, never safety I/O (those are unreachable
// here by construction). Every call is logged by the caller (§8.3).
METHOD ForceChannel : BOOL
VAR_INPUT
    ChannelPath : STRING(255);
    Force       : BOOL;     // TRUE = hold the value, FALSE = release
    BoolValue   : BOOL;     // digital output
    AnalogRaw   : DINT;     // analog output (raw)
END_VAR
END_METHOD

END_INTERFACE

// ---- Interfaces/I_Module.TcIO
// Core §3.2 — everything a parent needs to discover, monitor, and roll up a child.
// Reconciliation vs. Core §3.2 text: no ErrorID property here (it would collide with
// the PLCopen ErrorID output every module exposes, Core §6.1); callers read
// GetFaultSummary().ReasonCode. GetFaultSummary returns ST_Diagnostic (Core §8.8),
// Recipe changeover is a prepare/commit/abort transaction (Core §3.8).
INTERFACE I_Module EXTENDS __System.IQueryInterface

METHOD Cyclic : BOOL
END_METHOD

// recursive first-out walk (Core §8.2, §6.9)
METHOD GetFaultSummary : ST_Diagnostic
END_METHOD

// Load/validate into staging only; active ParCfg remains unchanged.
METHOD PrepareRecipe : BOOL
VAR_INPUT
    Model : ST_ModelId;
END_VAR
END_METHOD

// Infallible bounded publication after a successful PrepareRecipe.
METHOD CommitRecipe
END_METHOD

METHOD AbortRecipe
END_METHOD

PROPERTY FaultActive : BOOL
GET
END_GET
END_PROPERTY

PROPERTY ModuleType : E_ModuleType
GET
END_GET
END_PROPERTY

PROPERTY Name : STRING(80)
GET
END_GET
END_PROPERTY

PROPERTY State : E_ExecState
GET
END_GET
END_PROPERTY

END_INTERFACE

// ---- Interfaces/I_PartCarrier.TcIO
// Core §3.16.2 — source-agnostic part carrier (mirrors I_RecipeProvider).
INTERFACE I_PartCarrier

// FALSE => caller faults with CARRIER_READ_FAILED (Core §3.16.2)
METHOD ReadContext : BOOL
VAR_IN_OUT
    Ctx : ST_PartContext;
END_VAR
END_METHOD

// FALSE => caller faults with CARRIER_WRITE_FAILED; MUST precede EVENT_PART_PROCESSED
METHOD WriteResult : BOOL
VAR_INPUT
    Ctx : ST_PartContext;
END_VAR
END_METHOD

END_INTERFACE

// ---- Interfaces/I_SequenceHost.TcIO
// Core §6.7/§6.8 — the bridge from a separately-compiled sequence POU (SFC/ST/LD)
// to its owning module's protected framework services: step record, condition
// waits, run-style gate, part lifecycle, decisions, and completion/fault.
// FB_UnitBase implements it once; a sequence receives it at Setup. It carries
// framework plumbing ONLY — application decisions stay in the sequence's steps.
INTERFACE I_SequenceHost

// §6.5 step record (feeds the §6.9 walk and the §8.11.4 profiler)
METHOD M_SequenceSetStep
VAR_INPUT
    StepNo : INT;
    StepName : STRING(120);
    Awaits : I_Module;
    AwaitingLabel : STRING(120);
    Class : E_TimeClass;
    ExpectedTime : TIME;
END_VAR
END_METHOD

// §6.9(b) named plain-condition wait
METHOD M_SequenceAwait : BOOL
VAR_INPUT
    Idx : INT;
    Label : STRING(120);
    Ok : BOOL;
END_VAR
END_METHOD

// §3.4.2 run-style pacing gate
METHOD M_SequenceStepGate : BOOL
VAR_INPUT
    Steppable : BOOL;
END_VAR
END_METHOD

// §3.16.3 EVENT_PART_RECEIVED
METHOD M_SequencePartReceived : BOOL
END_METHOD

// §3.16.3 EVENT_PART_PROCESSING_STARTED
METHOD M_SequencePartStarted
END_METHOD

// §3.16.1 measured value
METHOD M_SequencePartRecord : BOOL
VAR_INPUT
    RecordName : STRING(64);
    Value : LREAL;
    Minimum : LREAL;
    Maximum : LREAL;
    Target : LREAL;
    EngUnit : STRING(16);
END_VAR
END_METHOD

// §3.16.3 EVENT_PART_PROCESSED (write-result-first; counts by verdict §8.11.2)
METHOD M_SequencePartProcessed : BOOL
VAR_INPUT
    Verdict : E_Verdict;
    Reason : E_Reason;
END_VAR
END_METHOD

// §8.11.2 carrier-less fallback counter
METHOD M_SequenceCountGood
END_METHOD

// §6.11 publish a decision request
METHOD M_SequenceAskDecision
VAR_INPUT
    Req : ST_DecisionRequest;
END_VAR
END_METHOD

// §6.11 consume the answer once (0 = none yet)
METHOD M_SequenceTakeDecision : INT
END_METHOD

// §6.11 withdraw an open request
METHOD M_SequenceClearDecision
END_METHOD

// §6.1 one-shot sequence completion (finite chains)
METHOD M_SequenceComplete
END_METHOD

// §8.11.1 cycle-complete marker; FALSE = stop granted (chain must not loop)
METHOD M_SequenceEndOfCycle : BOOL
END_METHOD

// §6.9 first-out fault from a step
METHOD M_SequenceFault
VAR_INPUT
    Reason : E_Reason;
    DescriptionKey : STRING(255);
END_VAR
END_METHOD

// §3.4 — TRUE while a Stop is requested and the sequence still runs. A chain
// polls this at its between-cycles wait so a stop need not ride out a phantom cycle.
METHOD M_SequenceStopPending : BOOL
END_METHOD

// §3.4/§8.11 — accept a pending Stop BETWEEN cycles: abandon the open cycle
// profile (no §8.11.1 cycle is counted for a wait-only fragment) and complete.
METHOD M_SequenceStopNow
END_METHOD

END_INTERFACE

// ---- Interfaces/I_RecipeProvider.TcIO
// Core §3.8 — pluggable recipe/type-data source. Implementations MUST validate
// completeness and SchemaVersion before filling ParCfg (migrate-or-fault; never partial).
INTERFACE I_RecipeProvider

// fills the caller's ParCfg; FALSE => caller faults with RECIPE_INVALID (Core §3.8)
METHOD Load : BOOL
VAR_INPUT
    ModelCode : STRING;
    RecipeKey : STRING;
    pParCfg : PVOID;
    Size    : UDINT;
END_VAR
END_METHOD

PROPERTY Ready : BOOL
GET
END_GET
END_PROPERTY

PROPERTY Source : E_RecipeSource
GET
END_GET
END_PROPERTY

END_INTERFACE

// ---- Interfaces/I_StationConfig.TcIO
// Core §3.8a — persistent STATION configuration (deployment-fixed, NOT model-keyed):
// MES endpoint, scanner baud, scale calibration, etc. Same injection shape as
// I_RecipeProvider so a module consumes config without embedding transport, and the
// framework ships a local default (FB_LocalStationConfig). Distinct from recipe data:
// station config does not change at changeover and is never bundled into a model recipe.
INTERFACE I_StationConfig

// fills the caller's StationCfg; FALSE => caller handles the miss (default = compiled)
METHOD Load : BOOL
VAR_INPUT
    Key   : STRING;
    pCfg  : PVOID;
    Size  : UDINT;
END_VAR
END_METHOD

// persist an edited StationCfg back (HMI/asset-system writes); FALSE = rejected
METHOD Store : BOOL
VAR_INPUT
    Key   : STRING;
    pCfg  : PVOID;
    Size  : UDINT;
END_VAR
END_METHOD

END_INTERFACE

// ---- Interfaces/I_Unit.TcIO
// Core §3.2 — mode-owning tier
INTERFACE I_Unit EXTENDS I_Module

// returns FALSE if the mode is unsupported (Core §3.4/§3.7)
METHOD SetMode : BOOL
VAR_INPUT
    Mode : E_Mode;
END_VAR
END_METHOD

METHOD Start : BOOL
END_METHOD

METHOD Stop : BOOL
END_METHOD

PROPERTY ModeActive : E_Mode
GET
END_GET
END_PROPERTY

END_INTERFACE

// ---- Interfaces/I_VerdictProvider.TcIO
// Annex C §C.1 / Annex E — optional per-cycle part-verdict hook (0 = none => always OK).
INTERFACE I_VerdictProvider

// TRUE = part OK; called once at the verdict step
METHOD Evaluate : BOOL
END_METHOD

// first NOK reason when Evaluate() = FALSE — same vocabulary as a fault (Core §8.8)
PROPERTY Reason : E_Reason
GET
END_GET
END_PROPERTY

END_INTERFACE

// ---- Connectivity/FB_LocalRecipeProvider.TcPOU
// Core §3.8 local provider. Validation is generic BECAUSE SchemaVersion is the
// first UINT of every ParCfg/record (§3.8): stored first-UINT must equal the
// target's initialized first-UINT, else Load = FALSE and the caller faults
// RECIPE_INVALID. Never a partial apply. Types stage through PrepareRecipe.
FUNCTION_BLOCK FB_LocalRecipeProvider IMPLEMENTS I_RecipeProvider
VAR
    _n    : INT;
    _models : ARRAY[1..PL_Fraktal.MAX_RECIPES] OF STRING(80);
    _keys   : ARRAY[1..PL_Fraktal.MAX_RECIPES] OF STRING(80);
    {attribute 'OPC.UA.DA' := '0'}
    _ptr  : ARRAY[1..PL_Fraktal.MAX_RECIPES] OF PVOID;
    _size : ARRAY[1..PL_Fraktal.MAX_RECIPES] OF UDINT;
END_VAR

// no cyclic body

METHOD Load : BOOL
VAR_INPUT
    ModelCode : STRING;
    RecipeKey : STRING;
    pParCfg : PVOID;
    Size    : UDINT;
END_VAR
VAR
    i, hit, fallback : INT;
    puT, puS : POINTER TO UINT;
END_VAR
Load := FALSE;
hit := 0;
fallback := 0;
FOR i := 1 TO _n DO
    IF (_keys[i] = RecipeKey) AND (_models[i] = ModelCode) THEN
        hit := i;
        EXIT;
    ELSIF (_keys[i] = RecipeKey) AND (_models[i] = '') THEN
        fallback := i;
    END_IF
END_FOR
IF hit = 0 THEN
    hit := fallback;
END_IF
IF (hit = 0) OR (pParCfg = 0) OR (_size[hit] <> Size) THEN
    RETURN;                                       // unknown/size mismatch -> caller faults (§3.8)
END_IF
puT := pParCfg;
puS := _ptr[hit];
IF puT^ <> puS^ THEN
    RETURN;                                       // SchemaVersion mismatch: migrate-or-fault (§3.8)
END_IF
MEMCPY(destAddr := pParCfg, srcAddr := _ptr[hit], n := Size);
Load := TRUE;
END_METHOD

// application wiring: one record per (ModelCode, RecipeKey); empty ModelCode is fallback.
METHOD Register : BOOL
VAR_INPUT
    ModelCode : STRING(80);
    RecipeKey : STRING(80);
    pData  : PVOID;
    Size   : UDINT;
END_VAR
VAR
    i : INT;
END_VAR
IF (_n >= PL_Fraktal.MAX_RECIPES) OR (pData = 0) OR (RecipeKey = '') THEN
    Register := FALSE;
    RETURN;
END_IF
FOR i := 1 TO _n DO
    IF (_models[i] = ModelCode) AND (_keys[i] = RecipeKey) THEN
        Register := FALSE;
        RETURN;
    END_IF
END_FOR
_n := _n + 1;
_models[_n] := ModelCode;
_keys[_n]   := RecipeKey;
_ptr[_n]  := pData;
_size[_n] := Size;
Register := TRUE;
END_METHOD

PROPERTY Ready : BOOL
GET
Ready := (_n > 0);
END_GET
END_PROPERTY

PROPERTY Source : E_RecipeSource
GET
Source := E_RecipeSource.LOCAL;
END_GET
END_PROPERTY

END_FUNCTION_BLOCK

// ---- Connectivity/FB_LocalStationConfig.TcPOU
// Core §3.8a — DEFAULT station-config provider: in-PLC PERSISTENT records, editable
// locally over OPC UA (§3.10). Remote sources (asset system, MES) substitute later
// through I_StationConfig without touching module code (O1, O6).
{attribute 'OPC.UA.DA' := '1'}
FUNCTION_BLOCK FB_LocalStationConfig IMPLEMENTS I_StationConfig
VAR PERSISTENT
    _n : INT;
END_VAR
VAR
    _keys : ARRAY[1..PL_Fraktal.MAX_STATIONCFG] OF STRING(80);
    _ptr  : ARRAY[1..PL_Fraktal.MAX_STATIONCFG] OF PVOID;
    _size : ARRAY[1..PL_Fraktal.MAX_STATIONCFG] OF UDINT;
END_VAR

// no cyclic body

METHOD Load : BOOL
VAR_INPUT
    Key : STRING;
    pCfg : PVOID;
    Size : UDINT;
END_VAR
VAR
    i : INT;
END_VAR
Load := FALSE;
FOR i := 1 TO _n DO
    IF (_keys[i] = Key) AND (_size[i] = Size) AND (pCfg <> 0) THEN
        MEMCPY(destAddr := pCfg, srcAddr := _ptr[i], n := Size);
        Load := TRUE;
        RETURN;
    END_IF
END_FOR
END_METHOD

METHOD Store : BOOL
VAR_INPUT
    Key : STRING;
    pCfg : PVOID;
    Size : UDINT;
END_VAR
VAR
    i : INT;
END_VAR
Store := FALSE;
FOR i := 1 TO _n DO
    IF (_keys[i] = Key) AND (_size[i] = Size) AND (pCfg <> 0) THEN
        MEMCPY(destAddr := _ptr[i], srcAddr := pCfg, n := Size);   // persists (registered targets live in persistent areas)
        Store := TRUE;
        RETURN;
    END_IF
END_FOR
END_METHOD

// application wiring: bind a module's PERSISTENT StationCfg to a key
METHOD Register : BOOL
VAR_INPUT
    Key : STRING(80);
    pData : PVOID;
    Size : UDINT;
END_VAR
IF (_n >= PL_Fraktal.MAX_STATIONCFG) OR (pData = 0) THEN
    Register := FALSE;
    RETURN;
END_IF
_n := _n + 1;
_keys[_n] := Key;
_ptr[_n] := pData;
_size[_n] := Size;
Register := TRUE;
END_METHOD

END_FUNCTION_BLOCK

// ---- Connectivity/FB_LocalAccessProvider.TcPOU
// Core §7.7(c) — DEFAULT local provider: persistent user/PIN table. Remote/central
// auth (server, LDAP via gateway) substitutes behind I_AccessProvider later.
FUNCTION_BLOCK FB_LocalAccessProvider IMPLEMENTS I_AccessProvider
VAR PERSISTENT
    _users : ARRAY[1..PL_Fraktal.MAX_USERS] OF ST_UserRecord;
    _n     : INT;
END_VAR

// no cyclic body

METHOD Authenticate : E_AccessLevel
VAR_INPUT
    User : STRING(32);
    Secret : STRING(32);
END_VAR
VAR
    i : INT;
END_VAR
Authenticate := E_AccessLevel.NONE;
FOR i := 1 TO _n DO
    IF (_users[i].User = User) AND (_users[i].Pin = Secret) THEN
        Authenticate := _users[i].Level;
        RETURN;
    END_IF
END_FOR
END_METHOD

// commissioning-time user entry (itself an ACCESS_POLICY-gated edit via the HMI).
// Idempotent by User: re-registering updates PIN/level (the table is PERSISTENT,
// so a composition root may register its defaults every boot without duplicates).
METHOD Register : BOOL
VAR_INPUT
    User : STRING(32);
    Pin : STRING(32);
    Level : E_AccessLevel;
END_VAR
VAR
    i : INT;
END_VAR
FOR i := 1 TO _n DO
    IF _users[i].User = User THEN
        _users[i].Pin   := Pin;
        _users[i].Level := Level;
        Register := TRUE;
        RETURN;
    END_IF
END_FOR
IF _n >= PL_Fraktal.MAX_USERS THEN
    Register := FALSE;
    RETURN;
END_IF
_n := _n + 1;
_users[_n].User  := User;
_users[_n].Pin   := Pin;
_users[_n].Level := Level;
Register := TRUE;
END_METHOD

END_FUNCTION_BLOCK

// ---- BaseClasses/FB_AccessManager.TcPOU
// Core §7.7(c) — per-root session + enforcement. Login/logout is DATA-DRIVEN
// (§3.10(a')): the HMI writes ReqUser/ReqSecret and pulses ReqLogin/ReqLogout;
// the secret is cleared after every attempt. Policy default: fully open (§7.7(b)).
{attribute 'OPC.UA.DA' := '1'}
FUNCTION_BLOCK FB_AccessManager
VAR_INPUT
    ReqUser   : STRING(32);          // HMI-writable login request
    ReqSecret : STRING(32);          // cleared after each attempt (§7.7(c))
    ReqLogin  : BOOL;
    ReqLogout : BOOL;
END_VAR
VAR_OUTPUT
    CurrentUser  : STRING(32);
    CurrentLevel : E_AccessLevel;    // HMI greys controls from this; PLC re-checks
    LoginFailed  : BOOL;             // last attempt outcome (HMI feedback)
END_VAR
VAR PERSISTENT
    Policy : ST_AccessPolicy;        // §3.8a station config; edit gated by ACCESS_POLICY
END_VAR
VAR
    _provider : I_AccessProvider;
    _log      : POINTER TO FB_AlarmLog;
    _tIdle    : TON;
END_VAR

// event/session handling is in Cyclic (called by the owning Unit each scan)

METHOD Cyclic : BOOL
VAR
    lvl : E_AccessLevel;
    loginHandled : BOOL;
    logoutHandled : BOOL;
END_VAR
loginHandled := ReqLogin;
IF loginHandled THEN
    ReqLogin := FALSE;
    lvl := E_AccessLevel.NONE;
    IF _provider <> 0 THEN
        lvl := _provider.Authenticate(User := ReqUser, Secret := ReqSecret);
    END_IF
    ReqSecret := '';                                   // never retain the secret
    IF lvl > E_AccessLevel.NONE THEN
        CurrentUser := ReqUser;
        CurrentLevel := lvl;
        LoginFailed := FALSE;
        _M_Audit('std.audit.login', CurrentUser);
    ELSE
        LoginFailed := TRUE;
        _M_Audit('std.audit.loginFailed', ReqUser);
    END_IF
END_IF
logoutHandled := ReqLogout;
IF logoutHandled THEN
    ReqLogout := FALSE;
    IF CurrentLevel > E_AccessLevel.NONE THEN
        _M_Audit('std.audit.logout', CurrentUser);
        CurrentUser := '';
        CurrentLevel := E_AccessLevel.NONE;
    END_IF
END_IF
// idle auto-logout (§7.7(c)); any successful login rearms it
_tIdle(IN := (Policy.SessionTimeout > T#0S) AND (CurrentLevel > E_AccessLevel.NONE) AND NOT loginHandled,
       PT := Policy.SessionTimeout);
IF _tIdle.Q THEN
    _M_Audit('std.audit.autoLogout', CurrentUser);
    CurrentUser := '';
    CurrentLevel := E_AccessLevel.NONE;
END_IF
Cyclic := TRUE;
END_METHOD

// Startup/station-configuration seam; runtime HMI writes remain Unit-gated.
METHOD ConfigureRequired : BOOL
VAR_INPUT
    Gate : E_GatedAction;
    Level : E_AccessLevel;
END_VAR
IF (TO_INT(Gate) < 0) OR (TO_INT(Gate) > TO_INT(E_GatedAction.POWER_CONTROL)) THEN
    ConfigureRequired := FALSE;
ELSE
    Policy.Required[TO_INT(Gate)] := Level;
    ConfigureRequired := TRUE;
END_IF
END_METHOD

// ST-facing request seam. OPC UA clients continue to write the published request data.
METHOD RequestLogin : BOOL
VAR_INPUT
    User : STRING(32);
    Secret : STRING(32);
END_VAR
ReqUser := User;
ReqSecret := Secret;
ReqLogin := TRUE;
RequestLogin := TRUE;
END_METHOD

// ST-facing request seam; the cyclic edge handler performs the state change and audit.
METHOD RequestLogout : BOOL
ReqLogout := TRUE;
RequestLogout := TRUE;
END_METHOD

// pure check for UI/logic — no logging
METHOD Permits : BOOL
VAR_INPUT
    Gate : E_GatedAction;
END_VAR
Permits := TO_DINT(CurrentLevel) >= TO_DINT(Policy.Required[TO_INT(Gate)]);
END_METHOD

// gated-entry check: a DENIED attempt is audited as a MESSAGE event (§8.3/§7.7(c))
METHOD PermitsLogged : BOOL
VAR_INPUT
    Gate : E_GatedAction;
END_VAR
PermitsLogged := Permits(Gate := Gate);
IF NOT PermitsLogged THEN
    _M_Audit('std.audit.accessDenied', CurrentUser);
END_IF
END_METHOD

METHOD Setup : BOOL
VAR_INPUT
    Provider : I_AccessProvider;
    pAlarmLog : POINTER TO FB_AlarmLog;
END_VAR
IF Provider <> 0 THEN
    _provider := Provider;                  // Unit OnInit may attach only the audit log
END_IF
_log := pAlarmLog;
Setup := TRUE;
END_METHOD

// audit trail for free: come+gone MESSAGE lands in the §8.3 ring
METHOD PRIVATE _M_Audit
VAR_INPUT
    What : STRING(64);
    Who : STRING(32);
END_VAR
VAR
    auditSlot : INT;
    txt : STRING(255);
END_VAR
IF _log = 0 THEN
    RETURN;
END_IF
txt := CONCAT(What, ': ');
txt := CONCAT(txt, Who);
auditSlot := _log^.Raise(Reason := E_Reason.NONE, Text := txt,
                 Source := 'Access', Severity := E_Severity.LOW,
                 Category := E_Category.SYSTEM, ResetClass := E_ResetClass.AUTO_RESET);
IF auditSlot > 0 THEN
    _log^.Gone(Slot := auditSlot);                     // instant come+gone -> ring entry
END_IF
END_METHOD

END_FUNCTION_BLOCK

// ---- BaseClasses/FB_AlarmLog.TcPOU
// Core §8.3 — per-Unit alarm & event log: active list + closed ring, durations,
// AUTO/MANUAL reset classes, optional historian sink. Fixed-size, never allocates.
{attribute 'OPC.UA.DA' := '1'}
FUNCTION_BLOCK FB_AlarmLog
VAR_OUTPUT
    Active    : ARRAY[1..PL_Fraktal.MAX_ALARM_ACTIVE] OF ST_AlarmEvent;  // ACTIVE/WAIT_RESET
    NActive   : INT;
    Ring      : ARRAY[1..PL_Fraktal.MAX_ALARM_RING] OF ST_AlarmEvent;    // closed, newest at RingHead
    RingHead  : INT;
    Blocking  : BOOL;    // any MANUAL_RESET event ACTIVE/WAIT_RESET (§8.3(b))
    Truncated : BOOL;
    Meta      : ARRAY[1..PL_Fraktal.MAX_ALARM_META] OF ST_AlarmMeta;  // §8.9 rationalization
    MetaCount : INT;
END_VAR
VAR
    _sink    : I_EventSink;
    _comeMs  : ARRAY[1..PL_Fraktal.MAX_ALARM_ACTIVE] OF DWORD;   // monotonic (TC3 §8.11)
    _shelfMs : ARRAY[1..PL_Fraktal.MAX_ALARM_ACTIVE] OF UDINT;   // §8.10 countdown (0 = not shelved)
    _cycLast : TIME;                                             // Cyclic delta stamp
END_VAR

// event-driven; no cyclic body

// §8.3(c) — open a non-channel-specific event; returns slot (0 = full).
METHOD Raise : INT
VAR_INPUT
    Reason : E_Reason;
    Text : STRING(255);
    Source : STRING(255);
    Severity : E_Severity;
    Category : E_Category;
    ResetClass : E_ResetClass;
END_VAR
Raise := _M_Raise(Reason := Reason, Text := Text, Source := Source,
    IoTag := '', IoAddress := '', Severity := Severity, Category := Category,
    ResetClass := ResetClass);
END_METHOD

// §8.3(c) — open an event; returns its slot id (0 = table full -> Truncated)
METHOD PRIVATE _M_Raise : INT
VAR_INPUT
    Reason : E_Reason;
    Text : STRING(255);
    Source : STRING(255);
    IoTag : STRING(80);
    IoAddress : STRING(80);
    Severity : E_Severity;
    Category : E_Category;
    ResetClass : E_ResetClass;
END_VAR
VAR
    i, slot : INT;
END_VAR
slot := 0;
FOR i := 1 TO PL_Fraktal.MAX_ALARM_ACTIVE DO
    IF Active[i].State = E_AlarmState.CLOSED THEN
        slot := i;
        EXIT;
    END_IF
END_FOR
IF slot = 0 THEN
    Truncated := TRUE;
    _M_Raise := 0;
    RETURN;
END_IF
Active[slot].ReasonCode  := Reason;
Active[slot].Description := Text;
Active[slot].SourcePath  := Source;
Active[slot].IoTag       := IoTag;
Active[slot].IoAddress   := IoAddress;
Active[slot].Severity    := Severity;
Active[slot].Category    := Category;
Active[slot].ResetClass  := ResetClass;
Active[slot].State       := E_AlarmState.ACTIVE;
Active[slot].ComeAt      := F_Now();
Active[slot].GoneAt      := DT#1970-01-01-00:00:00;
Active[slot].ResetAt     := DT#1970-01-01-00:00:00;
Active[slot].Duration    := T#0S;
Active[slot].Shelved     := FALSE;
Active[slot].ShelvedUntil:= DT#1970-01-01-00:00:00;
_shelfMs[slot] := 0;
_comeMs[slot] := TIME_TO_DWORD(TIME());
NActive := NActive + 1;
_M_UpdateBlocking();
IF _sink <> 0 THEN
    _sink.OnEvent(Ev := Active[slot]);              // come notification (§8.3(d))
END_IF
_M_Raise := slot;
END_METHOD

// §8.3(c) — open an ERROR event straight from a first-out diagnostic (no re-authoring)
METHOD RaiseDiag : INT
VAR_INPUT
    D : ST_Diagnostic;
    ResetClass : E_ResetClass;
END_VAR
RaiseDiag := _M_Raise(Reason := D.ReasonCode, Text := D.Description,
                   Source := D.SourcePath, IoTag := D.IoTag, IoAddress := D.IoAddress,
                   Severity := D.Severity, Category := D.Category,
                   ResetClass := ResetClass);
END_METHOD

// §8.3(b) — condition re-established: AUTO_RESET closes with Duration;
// MANUAL_RESET stays blocking in WAIT_RESET until OperatorReset.
METHOD Gone : BOOL
VAR_INPUT
    Slot : INT;
END_VAR
Gone := FALSE;
IF (Slot < 1) OR (Slot > PL_Fraktal.MAX_ALARM_ACTIVE) THEN
    RETURN;
END_IF
IF Active[Slot].State <> E_AlarmState.ACTIVE THEN
    RETURN;
END_IF
Active[Slot].GoneAt   := F_Now();
Active[Slot].Duration := DWORD_TO_TIME(TIME_TO_DWORD(TIME()) - _comeMs[Slot]);   // wrap-safe
IF Active[Slot].ResetClass = E_ResetClass.AUTO_RESET THEN
    _M_Close(Slot);
ELSE
    Active[Slot].State := E_AlarmState.WAIT_RESET;   // still blocking (§8.3(b))
END_IF
Gone := TRUE;
END_METHOD

// §8.3(b) — deliberate, release-gated operator action (§7.6/§14): closes
// MANUAL_RESET events whose condition is gone. NEVER self-invoked (§9.3 principle).
METHOD OperatorReset : BOOL
VAR
    i : INT;
END_VAR
OperatorReset := FALSE;
FOR i := 1 TO PL_Fraktal.MAX_ALARM_ACTIVE DO
    IF Active[i].State = E_AlarmState.WAIT_RESET THEN
        Active[i].ResetAt := F_Now();
        _M_Close(i);
        OperatorReset := TRUE;
    END_IF
END_FOR
END_METHOD

METHOD SetSink : BOOL
VAR_INPUT
    Sink : I_EventSink;
END_VAR
_sink := Sink;
SetSink := TRUE;
END_METHOD

METHOD PRIVATE _M_Close
VAR_INPUT
    Slot : INT;
END_VAR
Active[Slot].State := E_AlarmState.CLOSED;
RingHead := (RingHead MOD PL_Fraktal.MAX_ALARM_RING) + 1;
Ring[RingHead] := Active[Slot];
Ring[RingHead].State := E_AlarmState.CLOSED;
NActive := NActive - 1;
_M_UpdateBlocking();
IF _sink <> 0 THEN
    _sink.OnEvent(Ev := Ring[RingHead]);            // close notification with Duration (§8.3(d))
END_IF
END_METHOD

METHOD PRIVATE _M_UpdateBlocking
VAR
    i : INT;
    b : BOOL;
END_VAR
b := FALSE;
FOR i := 1 TO PL_Fraktal.MAX_ALARM_ACTIVE DO
    IF (Active[i].ResetClass = E_ResetClass.MANUAL_RESET)
    AND (Active[i].State <> E_AlarmState.CLOSED) THEN
        b := TRUE;
        EXIT;
    END_IF
END_FOR
Blocking := b;
END_METHOD

// §8.9 — register/update the rationalization record for a ReasonCode (idempotent).
// Modules/Units call at Setup. No record => the reason is NOT shelvable (§8.10).
METHOD RegisterMeta : BOOL
VAR_INPUT
    Reason         : E_Reason;
    OperatorAction : STRING(255);
    Consequence    : STRING(255);
    Shelvable      : BOOL;
END_VAR
VAR
    i : INT;
END_VAR
FOR i := 1 TO MetaCount DO
    IF Meta[i].ReasonCode = Reason THEN
        Meta[i].OperatorAction := OperatorAction;
        Meta[i].Consequence := Consequence;
        Meta[i].Shelvable := Shelvable;
        RegisterMeta := TRUE;
        RETURN;
    END_IF
END_FOR
IF MetaCount >= PL_Fraktal.MAX_ALARM_META THEN
    RegisterMeta := FALSE;
    RETURN;
END_IF
MetaCount := MetaCount + 1;
Meta[MetaCount].ReasonCode := Reason;
Meta[MetaCount].OperatorAction := OperatorAction;
Meta[MetaCount].Consequence := Consequence;
Meta[MetaCount].Shelvable := Shelvable;
RegisterMeta := TRUE;
END_METHOD

// §8.10 — may this active slot be shelved? SAFETY never; no meta record => no.
METHOD PROTECTED _M_Shelvable : BOOL
VAR_INPUT
    Slot : INT;
END_VAR
VAR
    i : INT;
END_VAR
_M_Shelvable := FALSE;
IF Slot < 1 OR Slot > PL_Fraktal.MAX_ALARM_ACTIVE THEN
    RETURN;
END_IF
IF Active[Slot].State = E_AlarmState.CLOSED THEN
    RETURN;
END_IF
IF Active[Slot].Category = E_Category.SAFETY THEN
    RETURN;                              // §8.10: safety never shelvable
END_IF
FOR i := 1 TO MetaCount DO
    IF Meta[i].ReasonCode = Active[Slot].ReasonCode THEN
        _M_Shelvable := Meta[i].Shelvable;
        RETURN;
    END_IF
END_FOR
// no rationalization record => not shelvable (rationalize first, §8.10)
END_METHOD

// §8.10 — suppress ANNUNCIATION of an active alarm for DurationS seconds (capped).
// Control is untouched: Blocking, interlocks, release reports all still see it.
// Caller has already checked §7.7 ALARM_SHELVE; the shelf itself is logged here.
METHOD Shelve : BOOL
VAR_INPUT
    Slot      : INT;
    DurationS : UDINT;
END_VAR
VAR
    auditSlot : INT;
END_VAR
IF NOT _M_Shelvable(Slot := Slot) THEN
    Shelve := FALSE;
    RETURN;
END_IF
IF DurationS = 0 THEN
    Shelve := FALSE;                              // every shelf is time-bounded
    RETURN;
END_IF
IF DurationS > PL_Fraktal.MAX_SHELF_S THEN
    DurationS := PL_Fraktal.MAX_SHELF_S;         // §8.10 time-bounded
END_IF
Active[Slot].Shelved := TRUE;
Active[Slot].ShelvedUntil := DWORD_TO_DT(DT_TO_DWORD(F_Now()) + DurationS);
_shelfMs[Slot] := DurationS * 1000;
auditSlot := Raise(Reason := E_Reason.NONE,
    Text := 'std.audit.alarmShelved', Source := Active[Slot].SourcePath,
    Severity := E_Severity.LOW, Category := E_Category.SYSTEM, ResetClass := E_ResetClass.AUTO_RESET);
IF auditSlot > 0 THEN Gone(Slot := auditSlot); END_IF
Shelve := TRUE;
END_METHOD

// §8.10 — restore annunciation (operator or auto-expiry). Logged.
METHOD Unshelve : BOOL
VAR_INPUT
    Slot : INT;
END_VAR
VAR
    auditSlot : INT;
END_VAR
IF Slot < 1 OR Slot > PL_Fraktal.MAX_ALARM_ACTIVE THEN
    Unshelve := FALSE;
    RETURN;
END_IF
IF NOT Active[Slot].Shelved THEN
    Unshelve := FALSE;
    RETURN;
END_IF
Active[Slot].Shelved := FALSE;
_shelfMs[Slot] := 0;
auditSlot := Raise(Reason := E_Reason.NONE,
    Text := 'std.audit.alarmUnshelved', Source := Active[Slot].SourcePath,
    Severity := E_Severity.LOW, Category := E_Category.SYSTEM, ResetClass := E_ResetClass.AUTO_RESET);
IF auditSlot > 0 THEN Gone(Slot := auditSlot); END_IF
Unshelve := TRUE;
END_METHOD

// §8.10 — auto-unshelve countdown (owning Unit ticks this each scan).
METHOD Cyclic : BOOL
VAR
    currentTime : TIME;
    deltaMs     : UDINT;
    i   : INT;
END_VAR
currentTime := TIME();                 // monotonic duration clock
IF _cycLast = T#0S THEN
    _cycLast := currentTime;
    Cyclic := TRUE;
    RETURN;
END_IF
deltaMs := TIME_TO_UDINT(currentTime) - TIME_TO_UDINT(_cycLast);
_cycLast := currentTime;
FOR i := 1 TO PL_Fraktal.MAX_ALARM_ACTIVE DO
    IF Active[i].Shelved AND _shelfMs[i] > 0 THEN
        IF _shelfMs[i] > deltaMs THEN
            _shelfMs[i] := _shelfMs[i] - deltaMs;
        ELSE
            _shelfMs[i] := 0;
            Unshelve(Slot := i);                 // §8.10 auto-expire (logged by Unshelve)
        END_IF
    END_IF
END_FOR
Cyclic := TRUE;
END_METHOD

END_FUNCTION_BLOCK

// ---- Platform/F_Now.TcPOU
// [TC3] Synchronized-clock read (Core §2.7 / TC3 §2.7). One clock feeds ALL
// timestamps (diagnostics §8.8, alarms §8.3, traceability §3.16, host events §11.6).
// Uses the TwinCAT system time (UTC). Validate against the pinned TwinCAT version.
FUNCTION F_Now : DT
VAR
    ft  : Tc2_Utilities.T_FILETIME64;  // 100 ns units since 1601-01-01 (UTC)
    sec : ULINT;
END_VAR

ft  := Tc2_Utilities.F_GetSystemTime();
sec := (ft - 116444736000000000) / 10000000;    // -> seconds since 1970-01-01 (UTC)
F_Now := DWORD_TO_DT(ULINT_TO_DWORD(sec));

END_FUNCTION

// ---- BaseClasses/FB_AsciiDeviceCM.TcPOU
// Core §3.15.1a — CM base for ASCII request/response devices over I_ByteChannel
// (vision sensors, code readers, gauges). One-outstanding-request state machine:
// SendRequest -> await terminated response -> _M_OnResponse hook; silence -> fault
// 10402. Written ONCE against the neutral seam: porting = swap the channel (O4/O8).
// Reconnect: bounded retry via the channel; link state published for Annex D facet.
{attribute 'OPC.UA.DA' := '1'}
FUNCTION_BLOCK ABSTRACT FB_AsciiDeviceCM EXTENDS FB_ControlModuleBase
VAR
    Host        : STRING(80);          // §3.8 config (per deployment)
    Port        : UINT;
    Terminator  : STRING(2) := '$R';   // CR default; device profile may override
    RespTimeout : TIME := T#2S;
    LinkState   : E_ByteChannelState;  // published (Annex D link facet)
    LastResponse: STRING(255);         // published (diagnosis)
END_VAR
VAR
    _chan     : I_ByteChannel;
    _rx       : STRING(255);
    _pending  : BOOL;                  // one outstanding request
    _tResp    : TON;
    _tRetry   : TON;
    _retryMs  : TIME := T#500MS;       // bounded backoff (doubles to 10s)
    _openTried : BOOL;                 // backoff spaces RE-tries; the first Open is immediate
END_VAR

;  // driven via Cyclic (base) -> OnCyclic below

// wire the transport + endpoint. Call from the profile's Setup after _M_SetName.
METHOD SetupDevice : BOOL
VAR_INPUT
    Chan : I_ByteChannel;
    DevHost : STRING(80);
    DevPort : UINT;
END_VAR
IF Chan = 0 OR DevHost = '' THEN
    _M_FaultN(PL_TcpDevReasons.DEV_CFG_INVALID, 'std.error.deviceConnectionNotConfigured');
    SetupDevice := FALSE;
    RETURN;
END_IF
_chan := Chan;
Host := DevHost;
Port := DevPort;
SetupDevice := TRUE;
END_METHOD

// channel management + RX framing. Profiles override _M_OnResponse, not this.
METHOD PROTECTED OnCyclic : DINT
VAR
    pos : INT;
    resp : STRING(255);
END_VAR
OnCyclic := SUPER^.OnCyclic();
IF _chan = 0 THEN
    RETURN;
END_IF
_chan.Tick();
LinkState := _chan.State();
CASE LinkState OF
    E_ByteChannelState.CLOSED:
        IF NOT _openTried THEN
            _openTried := TRUE;                    // first sight of CLOSED: connect NOW
            _chan.Open(Host := Host, Port := Port);
            LinkState := _chan.State();            // a synchronous transport is OPEN this scan
        ELSE
            _tRetry(IN := TRUE, PT := _retryMs);   // failed before: bounded backoff (§3.15.2 spirit)
            IF _tRetry.Q THEN
                _tRetry(IN := FALSE);
                _chan.Open(Host := Host, Port := Port);
                LinkState := _chan.State();
                IF _retryMs < T#10S THEN
                    _retryMs := _retryMs * 2;
                END_IF
            END_IF
        END_IF
    E_ByteChannelState.OPEN:
        _openTried := FALSE;
        _retryMs := T#500MS;
        _chan.Poll(Buffer := _rx);
        pos := FIND(_rx, Terminator);
        IF pos > 0 THEN
            resp := LEFT(_rx, pos - 1);
            _rx := DELETE(_rx, pos + LEN(Terminator) - 1, 1);
            _pending := FALSE;
            _tResp(IN := FALSE);
            LastResponse := resp;
            _M_OnResponse(Response := resp);
        ELSIF LEN(_rx) >= 250 THEN
            _rx := '';
            _M_FaultN(PL_TcpDevReasons.DEV_RX_OVERFLOW, 'std.error.deviceResponseOverflow');
        END_IF
    E_ByteChannelState.FAULT:
        IF _pending THEN
            _pending := FALSE;
            _tResp(IN := FALSE);
        END_IF
        _M_FaultN(PL_TcpDevReasons.DEV_CHANNEL_FAULT, 'std.error.transportChannelFault');
        _chan.Close();
ELSE
    _M_FaultN(PL_TcpDevReasons.DEV_CHANNEL_FAULT, 'std.error.byteChannelStateInvalid');
    _chan.Close();
END_CASE
// response timeout watch
_tResp(IN := _pending, PT := RespTimeout);
IF _tResp.Q THEN
    _pending := FALSE;
    _tResp(IN := FALSE);
    _M_FaultN(PL_TcpDevReasons.DEV_RESP_TIMEOUT, 'std.error.deviceResponseTimeout');
END_IF
END_METHOD

// issue one request (terminator appended). FALSE if not connected or one pending.
METHOD SendRequest : BOOL
VAR_INPUT
    Text : STRING(250);
END_VAR
// live channel state: the cached LinkState is one scan old and would reject a
// request issued in the same scan the transport opened.
IF _chan = 0 OR (_chan.State() <> E_ByteChannelState.OPEN) THEN
    _M_FaultN(PL_TcpDevReasons.DEV_NOT_CONNECTED, 'std.error.deviceNotConnected');
    SendRequest := FALSE;
    RETURN;
END_IF
IF _pending THEN
    SendRequest := FALSE;              // one-outstanding-request contract
    RETURN;
END_IF
_pending := _chan.Send(Text := CONCAT(Text, Terminator));
SendRequest := _pending;
END_METHOD

// profile hook: parse one terminated response. Raise DEV_PROTOCOL on garbage.
METHOD PROTECTED _M_OnResponse
VAR_INPUT
    Response : STRING(255);
END_VAR
;
END_METHOD

END_FUNCTION_BLOCK

// ---- BaseClasses/FB_ControlModuleBase.TcPOU
// Core §2.2 — leaf-tier semantic base. The shared PLCopen lifecycle lives in
// FB_ModuleBase; this type supplies only the Control Module tier identity.
FUNCTION_BLOCK ABSTRACT FB_ControlModuleBase EXTENDS FB_ModuleBase IMPLEMENTS I_ControlModule

PROPERTY ModuleType : E_ModuleType
GET
ModuleType := E_ModuleType.CONTROL_MODULE;
END_GET
END_PROPERTY

END_FUNCTION_BLOCK

// ---- BaseClasses/FB_ModuleBase.TcPOU
// Core §2.2 / §6.1 — the PLCopen lifecycle written ONCE (template method).
// A concrete type EXTENDS this base, declares its Command/HAL/ParCfg members, and
// overrides only _M_Dispatch (+ optionally hooks and recipe transaction methods).
// Edge handling, ExecState mapping, Execute-drop reset, ErrorID publication, and
// abort routing are inherited. Conformance rows T1/T4 (Core §5.7) are satisfied here
// and proven once in FB_Base_Tests.
{attribute 'OPC.UA.DA' := '1'}
FUNCTION_BLOCK ABSTRACT FB_ModuleBase IMPLEMENTS I_Module
VAR_INPUT
    Execute : BOOL;    // rising edge starts the command (Core §6.1)
    Abort   : BOOL;    // requests a controlled abort
END_VAR
VAR_OUTPUT
    Busy    : BOOL;
    Done    : BOOL;
    Error   : BOOL;
    Aborted : BOOL;
    ErrorID : DWORD;   // = TO_DWORD(first-out ReasonCode), Core §8.8
END_VAR
VAR_OUTPUT
    Status : ST_ModuleStatus;   // Core §3.10(a')/§6.9(a) — the OPC UA data mirror
    Timing : ST_ModuleTiming;   // Core §8.11.4(a) — per-command timing, captured here once
    Nameplate   : ST_Nameplate;  // §3.10.1 asset identity (set at Setup; empty = none)
    Catalog     : ARRAY[1..PL_Fraktal.MAX_CMD_CATALOG] OF ST_CommandInfo;  // §7.6.1 published command list
    CatalogCount: INT;
    Safety       : ST_SafetyStatus;       // §9 optional read-only safety facet (Present=FALSE if absent)
    ControlPower : ST_ControlPowerStatus; // §9 optional control/power facet
END_VAR
VAR
    _name  : STRING(80);
    _exec  : E_ExecState := E_ExecState.READY;
    _step  : INT;
    _diag  : ST_Diagnostic;
    _rTrig : R_TRIG;
    _abortErrTrig : R_TRIG;
    _initialized : BOOL;
    _prevExec   : E_ExecState;
    _manualCmd  : DINT;          // §7.6.1 pending manual command value (0 = none)
    _manualReq  : BOOL;
    _manualActive : BOOL;        // one-shot manual request owns Execute until terminal state
    _cmdArmed   : BOOL;          // terminal state came from a command; gates the §6.1 reset
    _cmdId      : DINT;          // set by _M_TagCommand (one line per type, §8.11.4(a))
    _cmdLabel   : STRING(120);
    _tCmdStart  : DWORD;         // monotonic ms at command start (TC3 §8.11)
END_VAR

// FB body just runs the lifecycle; parents may call the instance or Cyclic() (I_Module)
Cyclic();

// Core §6.1 — edge -> hooks -> dispatch -> map -> Execute-drop reset
METHOD Cyclic : BOOL
// Execute-drop reset (Core §6.1): a COMMAND-produced terminal state published in
// an earlier scan plus Execute low resets to READY BEFORE this scan's mapping, so
// the outputs go idle in the same call. A completion later this scan still maps
// its one-cycle DONE/ERROR/ABORTED pulse first (PLCopen). Faults raised OUTSIDE a
// command (recipe/config at Setup, cyclic condition monitors) latch (§3.8/§8.3):
// Execute was never high, so the handshake reset does not consume them.
IF (NOT Execute) AND _cmdArmed
AND ((_exec = E_ExecState.DONE) OR (_exec = E_ExecState.ERROR) OR (_exec = E_ExecState.ABORTED)) THEN
    _exec := E_ExecState.READY;
    _cmdArmed := FALSE;
END_IF

_rTrig(CLK := Execute);
// A fresh command edge may also RETRY from a latched non-command fault: the edge
// clears the diagnostic and re-runs validation, which re-faults if the cause remains.
IF _rTrig.Q AND ((_exec = E_ExecState.READY)
    OR ((_exec = E_ExecState.ERROR) AND NOT _cmdArmed)) THEN
    _exec := E_ExecState.BUSY;      // ParCmd of the concrete type is latched on this edge
    _cmdArmed := TRUE;
    _step := 10;
    _M_ClearDiag();
    _tCmdStart := TIME_TO_DWORD(TIME());          // §8.11.4(a) command-timing start
END_IF

IF NOT _initialized THEN
    _initialized := TRUE;
    OnInit();                        // Core §3.14 one-shot for every module tier
END_IF
OnCyclic();                          // Core §3.14 hook: background management, no outputs

IF Abort AND (_exec = E_ExecState.BUSY) THEN
    OnAbort();                       // Core §3.14 hook: device-safe abort action
END_IF
_abortErrTrig(CLK := Abort AND (_exec = E_ExecState.ERROR));
IF _abortErrTrig.Q THEN
    OnAbortInError();                // distinct recovery hook; ERROR remains latched
END_IF

IF _exec = E_ExecState.BUSY THEN
    _M_Dispatch();                   // the ONLY thing a type must write (Core §2.2)
END_IF

// §8.11.4(a) — close the command's timing row on leaving BUSY (DONE/ERROR/ABORTED)
IF (_prevExec = E_ExecState.BUSY) AND (_exec <> E_ExecState.BUSY) THEN
    _M_RecordCmdTiming(TIME_TO_DWORD(TIME()) - _tCmdStart);   // wrap-safe diff (TC3 §8.11)
END_IF
_prevExec := _exec;

Busy    := (_exec = E_ExecState.BUSY);
Done    := (_exec = E_ExecState.DONE);
Error   := (_exec = E_ExecState.ERROR);
Aborted := (_exec = E_ExecState.ABORTED);
ErrorID := TO_DWORD(_diag.ReasonCode);

// §6.9(a)/§3.10(a') — refresh the data mirror: properties are invisible to the
// OPC UA namespace, so everything the HMI binds is published here as DATA
Status.ModuleType  := ModuleType;
Status.State       := _exec;
Status.FaultActive := (_exec = E_ExecState.ERROR);
Status.Diagnostic  := _diag;
_M_PublishStatus();              // tier-specific overlay after the common mirror is final

// A manual command is a one-shot use of the same PLCopen lifecycle. Keep the
// terminal state visible for this scan, then drop Execute for next-scan reset.
IF _manualActive AND ((_exec = E_ExecState.DONE) OR (_exec = E_ExecState.ERROR) OR (_exec = E_ExecState.ABORTED)) THEN
    Execute := FALSE;
    _manualActive := FALSE;
END_IF
Cyclic := TRUE;
END_METHOD

// Core §8.2/§6.9 — this node's first-out (composites override via rollup in the EM base)
METHOD GetFaultSummary : ST_Diagnostic
GetFaultSummary := _diag;
END_METHOD

// Core §3.14 hook — optional override: device-safe abort action.
// Override contract (Core §3.14.2): call SUPER^.OnAbort() FIRST and keep its return.
METHOD PROTECTED OnAbort : DINT
_exec := E_ExecState.ABORTED;
_step := 0;
OnAbort := 0;
END_METHOD

// Core §3.14 — optional error-state abort/recovery action. ERROR remains latched
// until Execute drops. Overrides call SUPER^.OnAbortInError() first.
METHOD PROTECTED OnAbortInError : DINT
OnAbortInError := 0;
END_METHOD

// Core §3.14 — first operational scan, after Setup/recipe load.
// Overrides call SUPER^.OnInit() first and propagate its return.
METHOD PROTECTED OnInit : DINT
OnInit := 0;
END_METHOD

// Core §3.14 hook — optional override: per-scan background management (idempotent,
// no direct outputs). Override contract: call SUPER^.OnCyclic() FIRST, keep return.
METHOD PROTECTED OnCyclic : DINT
OnCyclic := 0;
END_METHOD

// Core §3.8 — types with ParCfg load into staging here.
METHOD PrepareRecipe : BOOL
VAR_INPUT
    Model : ST_ModelId;
END_VAR
PrepareRecipe := TRUE;
END_METHOD

METHOD CommitRecipe
END_METHOD

METHOD AbortRecipe
END_METHOD

// Core §3.2 — generic DINT command path; the catalog is the supported set.
// Concrete dispatch consumes the inherited manual request, so typed/generic/HMI
// paths share validation, timing, interlocks, and the PLCopen lifecycle.
METHOD ExecuteCommand : BOOL
VAR_INPUT
    Command : DINT;
END_VAR
ExecuteCommand := ManualCommand(Value := Command);
END_METHOD

// Core §3.2/§6.1 — method form of the inherited abort route.
METHOD AbortCommand : BOOL
AbortCommand := FALSE;
IF _exec <> E_ExecState.BUSY THEN
    RETURN;
END_IF
OnAbort();
_exec := E_ExecState.ABORTED;
_step := 0;
AbortCommand := TRUE;
END_METHOD

METHOD PROTECTED _M_ClearDiag
_diag.ReasonCode  := E_Reason.NONE;
_diag.Description := '';
_diag.IoTag := '';
_diag.IoAddress := '';
END_METHOD

// Core §6.1 — successful completion (the concrete type publishes OutCmd before calling)
METHOD PROTECTED _M_Complete
_exec := E_ExecState.DONE;
_step := 0;
_M_ClearDiag();
END_METHOD

// Core §2.2 — THE extension point: the type's CASE _step device logic,
// calling _M_Fault / _M_FaultDiag / _M_Complete.
METHOD PROTECTED ABSTRACT _M_Dispatch
END_METHOD

// Core §6.9 — stamp the first-out reason and hold in ERROR
METHOD PROTECTED _M_Fault
VAR_INPUT
    Reason : E_Reason;
    Text   : STRING(255);
END_VAR
_diag.ReasonCode  := Reason;
_diag.Description := Text;
_diag.SourcePath  := _name;
_diag.IoTag       := '';
_diag.IoAddress   := '';
_diag.Severity    := E_Severity.MED;
_diag.Category    := E_Category.PROCESS;
_diag.Since       := F_Now();       // synchronized clock (Core §2.7)
_exec := E_ExecState.ERROR;
_step := 0;
END_METHOD

// Core §8.2 — adopt a ready-made diagnostic verbatim (rollup / connector reason)
METHOD PROTECTED _M_FaultDiag
VAR_INPUT
    Diag : ST_Diagnostic;
END_VAR
_diag := Diag;
_exec := E_ExecState.ERROR;
_step := 0;
END_METHOD

// called from the concrete type's Setup (Core §3.11); Name = browse path (Core §4.8)
METHOD PROTECTED _M_SetName
VAR_INPUT
    Name : STRING(80);
END_VAR
_name := Name;
Status.Name := Name;   // mirror (§3.10(a'))
END_METHOD

// Core §8.11.4(a) — fold the finished command into its timing row (find-or-allocate)
METHOD PRIVATE _M_RecordCmdTiming
VAR_INPUT
    DurMs : DWORD;
END_VAR
VAR
    i, slot : INT;
END_VAR
Timing.LastCmdTime := DWORD_TO_TIME(DurMs);
slot := 0;
FOR i := 1 TO PL_Fraktal.MAX_CMD_STATS DO
    IF (Timing.Rows[i].Count > 0) AND (Timing.Rows[i].Id = _cmdId) THEN
        slot := i;
        EXIT;
    ELSIF (slot = 0) AND (Timing.Rows[i].Count = 0) THEN
        slot := i;
    END_IF
END_FOR
IF slot = 0 THEN
    Timing.Truncated := TRUE;        // fixed array, never grown at runtime (§8.11.4(e))
ELSE
    Timing.Rows[slot].Id    := _cmdId;
    Timing.Rows[slot].Label := _cmdLabel;
    F_TimingUpdate(Row := Timing.Rows[slot], DurMs := DurMs);
END_IF
END_METHOD

// Core §8.11.4(a) — the ONE line a type adds for a per-command breakdown:
//   _M_TagCommand(TO_DINT(Command), '<label>');   (idempotent; scaffold includes it)
METHOD PROTECTED _M_TagCommand
VAR_INPUT
    Id    : DINT;
    Label : STRING(120);
END_VAR
_cmdId    := Id;
    _cmdLabel := Label;
END_METHOD

// Optional localizable HMI metadata; keys only, never operator prose.
METHOD PROTECTED _M_SetPresentation
VAR_INPUT
    DisplayNameKey : STRING(160);
    DescriptionKey : STRING(160);
END_VAR
Status.DisplayNameKey := DisplayNameKey;
Status.DescriptionKey := DescriptionKey;
END_METHOD

// Core §8.8 band-extensibility: fault with a per-type band code (DINT constant).
// E_Reason is deliberately non-strict, so the numeric assignment is contract, not a cast trick.
METHOD PROTECTED _M_FaultN
VAR_INPUT
    Code : DINT;          // registered band code (Core §8.8 registry)
    Text : STRING(255);
END_VAR
_diag.ReasonCode  := Code;    // non-strict enum accepts the band value (Core §8.8)
_diag.Description := Text;
_diag.SourcePath  := _name;
_diag.IoTag       := '';
_diag.IoAddress   := '';
_diag.Severity    := E_Severity.MED;
_diag.Category    := E_Category.PROCESS;
_diag.Since       := F_Now();
_exec := E_ExecState.ERROR;
_step := 0;
END_METHOD

// Type-band fault with the implicated schematic tag and terminal location.
METHOD PROTECTED _M_FaultIoN
VAR_INPUT
    Code : DINT;
    Text : STRING(255);
    IoTag : STRING(80);
    IoAddress : STRING(80);
END_VAR
_M_FaultN(Code := Code, Text := Text);
_diag.IoTag := IoTag;
_diag.IoAddress := IoAddress;
END_METHOD

PROPERTY FaultActive : BOOL
GET
FaultActive := (_exec = E_ExecState.ERROR);
END_GET
END_PROPERTY

PROPERTY ModuleType : E_ModuleType
GET
ModuleType := E_ModuleType.NONE;
END_GET
END_PROPERTY

PROPERTY Name : STRING(80)
GET
Name := _name;
END_GET
END_PROPERTY

PROPERTY State : E_ExecState
GET
State := _exec;
END_GET
END_PROPERTY

// §7.6.1 — register one manual command in the catalog (call in the module's init).
// Idempotent by Value: re-publishing a Value updates its label.
METHOD PROTECTED _M_PublishCommand
VAR_INPUT
    Value : DINT;
    Label : STRING(120);
END_VAR
VAR
    i : INT;
END_VAR
FOR i := 1 TO CatalogCount DO
    IF Catalog[i].Value = Value THEN
        Catalog[i].Label := Label;
        RETURN;
    END_IF
END_FOR
IF CatalogCount >= PL_Fraktal.MAX_CMD_CATALOG THEN
    RETURN;
END_IF
CatalogCount := CatalogCount + 1;
Catalog[CatalogCount].Value := Value;
Catalog[CatalogCount].Label := Label;
END_METHOD

// §7.6.1 — apply a manual command, routed THROUGH the normal command surface so
// interlocks/first-out/timing still apply (§3.2). The owning Unit is the single
// gate: it calls this ONLY after verifying MANUAL mode (§3.4) + MANUAL access
// (§7.7) and logs the §8.3 event. §7.6 Release<Function> is enforced by the
// module's own _M_Dispatch. Concrete modules read _manualReq/_manualCmd there.
METHOD ManualCommand : BOOL
VAR_INPUT
    Value : DINT;
END_VAR
VAR
    i : INT;
    supported : BOOL;
END_VAR
ManualCommand := FALSE;
FOR i := 1 TO CatalogCount DO
    IF Catalog[i].Value = Value THEN
        supported := TRUE;
        EXIT;
    END_IF
END_FOR
IF NOT supported THEN
    RETURN;                              // reject values outside the published set (§5.6)
END_IF
IF (_exec <> E_ExecState.READY) OR Execute OR _manualActive THEN
    RETURN;
END_IF
_manualCmd := Value;
_manualReq := TRUE;                       // consumed by the module's _M_Dispatch
_manualActive := TRUE;
Execute := TRUE;                          // rising edge enters the inherited lifecycle
ManualCommand := TRUE;
END_METHOD

// Called after the common Status mirror refresh. Derived tiers may overlay data.
METHOD PROTECTED _M_PublishStatus
;
END_METHOD

// §3.10.1 — set the module's asset identity once, at Setup. Not HMI-writable;
// identity, not configuration (deliberately outside §3.8/§7.7).
METHOD SetNameplate : BOOL
VAR_INPUT
    Plate : ST_Nameplate;
END_VAR
Nameplate := Plate;
SetNameplate := TRUE;
END_METHOD

END_FUNCTION_BLOCK

// ---- Platform/F_TimingUpdate.TcPOU
// Core §8.11.4 — fold one duration into a timing row: Count/Last/Min/Max and a
// running mean (avg += (x - avg)/n). Pure function so the math is testable exactly.
FUNCTION F_TimingUpdate : BOOL
VAR_IN_OUT
    Row : ST_TimingRow;
END_VAR
VAR_INPUT
    DurMs : DWORD;    // wrap-safe monotonic difference (TC3 §8.11)
END_VAR
VAR
    d, avg : DINT;
END_VAR

Row.Count := Row.Count + 1;
Row.Last  := DWORD_TO_TIME(DurMs);
IF (Row.Count = 1) OR (Row.Last < Row.Minimum) THEN
    Row.Minimum := Row.Last;
END_IF
IF Row.Last > Row.Maximum THEN
    Row.Maximum := Row.Last;
END_IF
d   := DWORD_TO_DINT(DurMs);
avg := TIME_TO_DINT(Row.Avg);
avg := avg + ((d - avg) / UDINT_TO_DINT(Row.Count));
Row.Avg := DINT_TO_TIME(avg);
F_TimingUpdate := TRUE;

END_FUNCTION

// ---- BaseClasses/FB_CycleProfiler.TcPOU
// Core §8.11.4(b)/(f) — the cycle-time profile, fed by the step record the chain
// already keeps for §6.9: StepChanged() from _M_SetStep (with the step's time class,
// WORK by default), CycleComplete() at the finish step (§8.11.1 marker). Application
// steps add NOTHING except one enum on genuine wait steps. The step-chain / Unit
// base (M2) calls both automatically; until then a Unit wires the two calls once
// (Annex C §C.6). Fixed-size, no runtime allocation (Core §8.11.4(e)).
{attribute 'OPC.UA.DA' := '1'}
FUNCTION_BLOCK FB_CycleProfiler
VAR_OUTPUT
    Current        : ST_CycleProfile;   // cycle in progress (live waterfall)
    LastCycle      : ST_CycleProfile;   // last completed cycle — the HMI chart source
    StepStats      : ARRAY[1..PL_Fraktal.MAX_PROFILE_STEPS] OF ST_TimingRow;  // per-StepNo aggregates
    StatsTruncated : BOOL;
    // §8.11.1 throughput markers + §8.11.4 trend ring (the cycle-time ANALYSIS source:
    // per-cycle work/wait-class totals, charted by the HMI to explain increases)
    LastCycleTime  : TIME;
    MinCycleTime   : TIME;              // rolling minimum since reset (the demonstrated best)
    History        : ARRAY[1..PL_Fraktal.MAX_CYCLE_HISTORY] OF ST_CycleSummary;
    HistoryHead    : INT;               // newest entry (0 = none yet)
    // §8.11.4(d) — degradation is data: WorkTime drifting beyond Baseline*(1+BandPct)
    // pulses DegradedTrig for ONE call so the owner raises the maintenance event once.
    BaselineWorkMs : UDINT;             // 0 = degradation watch off (§3.8 config)
    DegradedBandPct: UDINT := 20;       // allowed drift above baseline, percent
    DegradedTrig   : BOOL;
    DegradedWorkMs : UDINT;             // the WorkTime that tripped the band (for the event text)
END_VAR
VAR
    _running      : BOOL;
    _openNo       : INT;
    _openName     : STRING(80);
    _openClass    : E_TimeClass;
    _openExpected : TIME;
    _openStartMs  : DWORD;
    _openStartDt  : DT;
    _cycleStartMs : DWORD;
    _degraded     : BOOL;               // latched: one event per excursion, not per cycle
END_VAR

// no cyclic body — event-driven via StepChanged/CycleComplete

// close the open step and publish the cycle (call at the finish step, §8.11.1).
// Publishes WorkTime = ByClass[WORK] — the real cycle time (§8.11.4(f)).
METHOD CycleComplete : BOOL
VAR
    nowMs : DWORD;
END_VAR
IF NOT _running THEN
    CycleComplete := FALSE;
    RETURN;
END_IF
nowMs := TIME_TO_DWORD(TIME());
_M_CloseOpen(nowMs);
Current.Total    := DWORD_TO_TIME(nowMs - _cycleStartMs);   // wrap-safe (TC3 §8.11)
Current.WorkTime := Current.ByClass[TO_INT(E_TimeClass.WORK)];
Current.WaitTime := Current.Total - Current.WorkTime;
Current.CycleNo  := LastCycle.CycleNo + 1;
LastCycle := Current;

// §8.11.1 throughput markers
LastCycleTime := Current.Total;
IF (MinCycleTime = T#0S) OR (Current.Total < MinCycleTime) THEN
    MinCycleTime := Current.Total;
END_IF

// §8.11.4 trend ring — per-cycle class split for the HMI's cause analysis
HistoryHead := (HistoryHead MOD PL_Fraktal.MAX_CYCLE_HISTORY) + 1;
History[HistoryHead].CycleNo  := Current.CycleNo;
History[HistoryHead].Started  := Current.Started;
History[HistoryHead].Total    := Current.Total;
History[HistoryHead].WorkTime := Current.WorkTime;
History[HistoryHead].WaitTime := Current.WaitTime;
History[HistoryHead].ByClass  := Current.ByClass;

// §8.11.4(d) — degradation watch on WORK time (waits are attributed, not drift).
// One-call trigger, latched per excursion; recovery below the band rearms it.
DegradedTrig := FALSE;
DegradedWorkMs := TIME_TO_DWORD(Current.WorkTime);
IF BaselineWorkMs > 0 THEN
    IF DegradedWorkMs * 100 > BaselineWorkMs * (100 + DegradedBandPct) THEN
        IF NOT _degraded THEN
            _degraded := TRUE;
            DegradedTrig := TRUE;
        END_IF
    ELSE
        _degraded := FALSE;
    END_IF
END_IF

_running := FALSE;
_openNo  := 0;
CycleComplete := TRUE;
END_METHOD

// §8.11.1 — discard the OPEN cycle without publishing it: a stop accepted at the
// between-cycles wait must not count a wait-only fragment as a production cycle
// (it would poison MinCycleTime and the trend). Aggregates keep completed cycles.
METHOD CycleAbandon : BOOL
_running := FALSE;
_openNo := 0;
CycleAbandon := TRUE;
END_METHOD

// deliberate, LOGGED action only (Core §8.11.2) — the caller raises the event
METHOD ResetStats : BOOL
VAR
    i     : INT;
    empty : ST_TimingRow;
    emptySummary : ST_CycleSummary;
END_VAR
FOR i := 1 TO PL_Fraktal.MAX_PROFILE_STEPS DO
    StepStats[i] := empty;
END_FOR
FOR i := 1 TO PL_Fraktal.MAX_CYCLE_HISTORY DO
    History[i] := emptySummary;
END_FOR
HistoryHead := 0;
LastCycleTime := T#0S;
MinCycleTime := T#0S;
_degraded := FALSE;
StatsTruncated := FALSE;
LastCycle.CycleNo := 0;
ResetStats := TRUE;
END_METHOD

// Configure the recipe-owned WORK-time reference through the profiler owner.
// BaselineWorkMs is published read-only; TwinCAT therefore rejects assignment
// through a parent FB's published Profiler output. Zero disables the watch.
METHOD M_SetBaselineWork : BOOL
VAR_INPUT
    WorkMs : UDINT;
END_VAR
BaselineWorkMs := WorkMs;
DegradedTrig := FALSE;
_degraded := FALSE;
M_SetBaselineWork := TRUE;
END_METHOD

// call on every step change — _M_SetStep already has StepNo/StepName (§6.5).
// Class defaults to WORK; only genuine wait steps pass a wait class (§8.11.4(f)).
METHOD StepChanged : BOOL
VAR_INPUT
    StepNo   : INT;
    StepName : STRING(120);
    Class    : E_TimeClass;
    Expected : TIME;                   // §8.11.4(c) — declared guard, drawn vs actual
END_VAR
VAR
    nowMs : DWORD;
    i     : INT;
END_VAR
IF _running AND (StepNo = _openNo) THEN
    _openClass := Class;               // same step refreshed — class may be (re)declared
    _openExpected := Expected;
    StepChanged := TRUE;
    RETURN;
END_IF
nowMs := TIME_TO_DWORD(TIME());
IF NOT _running THEN
    _running := TRUE;                  // first step opens the cycle (§8.11.1 start marker)
    _cycleStartMs := nowMs;
    Current.Started   := F_Now();
    Current.NSteps    := 0;
    Current.Truncated := FALSE;
    FOR i := 0 TO 4 DO
        Current.ByClass[i] := T#0S;    // reset the class split for the new cycle
    END_FOR
ELSE
    _M_CloseOpen(nowMs);
END_IF
_openNo      := StepNo;
_openName    := StepName;
_openClass   := Class;
_openExpected := Expected;
_openStartMs := nowMs;
_openStartDt := F_Now();
StepChanged := TRUE;
END_METHOD

// fold the open step into the profile, the class split, and the aggregates
METHOD PRIVATE _M_CloseOpen
VAR_INPUT
    NowMs : DWORD;
END_VAR
VAR
    dur  : DWORD;
    i    : INT;
    slot : INT;
END_VAR
IF _openNo = 0 THEN
    RETURN;
END_IF
dur := NowMs - _openStartMs;                                // wrap-safe (TC3 §8.11)

// (1) ordered waterfall entry
IF Current.NSteps < PL_Fraktal.MAX_PROFILE_STEPS THEN
    Current.NSteps := Current.NSteps + 1;
    Current.Steps[Current.NSteps].StepNo   := _openNo;
    Current.Steps[Current.NSteps].StepName := _openName;
    Current.Steps[Current.NSteps].Class    := _openClass;
    Current.Steps[Current.NSteps].Started  := _openStartDt;
    Current.Steps[Current.NSteps].Duration := DWORD_TO_TIME(dur);
    Current.Steps[Current.NSteps].Expected := _openExpected;
ELSE
    Current.Truncated := TRUE;
END_IF

// (2) time-class split (§8.11.4(f)) — WorkTime/WaitTime derive from this at cycle close
Current.ByClass[TO_INT(_openClass)] := Current.ByClass[TO_INT(_openClass)] + DWORD_TO_TIME(dur);

